   VAR
      sUDT_CommonStatus { ExternalAccessible := 'False'; ExternalVisible := 'False'; ExternalWritable := 'False'; S7_SetPoint := 'False'} : "UDT_CommonStatus";   // Common status structure
      sUDT_CommonStatusOld { ExternalAccessible := 'False'; ExternalVisible := 'False'; ExternalWritable := 'False'; S7_SetPoint := 'False'} : "UDT_CommonStatus";   // Auxiliary status structure
      sUDT_HMIStatus { ExternalAccessible := 'False'; ExternalVisible := 'False'; ExternalWritable := 'False'; S7_SetPoint := 'False'} : "UDT_CaljanStatus";   // HMI status structure
      sUDT_PNDevice { ExternalAccessible := 'False'; ExternalVisible := 'False'; ExternalWritable := 'False'; S7_SetPoint := 'False'} : "UDT_PNDevice";   // PN device info structure
      sa_PNPortsStatus { ExternalAccessible := 'False'; ExternalVisible := 'False'; ExternalWritable := 'False'} : Array[1..8] of Bool;   // TRUE when specific port has an error
      R_TRIG_EnergySave {InstructionName := 'R_TRIG'; LibVersion := '1.0'; ExternalAccessible := 'False'; ExternalVisible := 'False'; ExternalWritable := 'False'; S7_SetPoint := 'False'} : R_TRIG;   // Rising edge for energy save
      R_TRIG_ConveyorUp {InstructionName := 'R_TRIG'; LibVersion := '1.0'; ExternalAccessible := 'False'; ExternalVisible := 'False'; ExternalWritable := 'False'; S7_SetPoint := 'False'} : R_TRIG;   // Rising edge of automatic active
      R_TRIG_ConveyorDown {InstructionName := 'R_TRIG'; LibVersion := '1.0'; ExternalAccessible := 'False'; ExternalVisible := 'False'; ExternalWritable := 'False'; S7_SetPoint := 'False'} : R_TRIG;   // Rising edge of automatic not active
      R_TRIG_NotHealthy {InstructionName := 'R_TRIG'; LibVersion := '1.0'; ExternalAccessible := 'False'; ExternalVisible := 'False'; ExternalWritable := 'False'; S7_SetPoint := 'False'} : R_TRIG;   // Rising edge trigger if extendable not healthy
      R_TRIG_TooLongParcel {InstructionName := 'R_TRIG'; LibVersion := '1.0'; ExternalAccessible := 'False'; ExternalVisible := 'False'; ExternalWritable := 'False'; S7_SetPoint := 'False'} : R_TRIG;   // Rising edge trigger for too long parcel
      R_TRIG_SafetyOk {InstructionName := 'R_TRIG'; LibVersion := '1.0'; ExternalAccessible := 'False'; ExternalVisible := 'False'; ExternalWritable := 'False'; S7_SetPoint := 'False'} : R_TRIG;   // Rising edge trigger safety is ok
      R_TRIG_PEC_UnloaderFiltered {InstructionName := 'R_TRIG'; LibVersion := '1.0'; ExternalAccessible := 'False'; ExternalVisible := 'False'; ExternalWritable := 'False'; S7_SetPoint := 'False'} : R_TRIG;   // Rising edge trigger end of section photo eye filtered
      F_TRIG_PEC_UnloaderFiltered {InstructionName := 'F_TRIG'; LibVersion := '1.0'; ExternalAccessible := 'False'; ExternalVisible := 'False'; ExternalWritable := 'False'; S7_SetPoint := 'False'} : F_TRIG;   // Falling edge trigger end of section photo eye filtered
      F_TRIG_AuxHeadToEnd {InstructionName := 'F_TRIG'; LibVersion := '1.0'; ExternalAccessible := 'False'; ExternalVisible := 'False'; ExternalWritable := 'False'; S7_SetPoint := 'False'} : F_TRIG;   // Falling edge trigger Aux head to end bit
      R_TRIG_TailToBegin {InstructionName := 'R_TRIG'; LibVersion := '1.0'; ExternalAccessible := 'False'; ExternalVisible := 'False'; ExternalWritable := 'False'; S7_SetPoint := 'False'} : R_TRIG;   // Rising edge trigger tail to begin bit
      sR_TRIG_PNSlaveError {InstructionName := 'R_TRIG'; LibVersion := '1.0'; ExternalAccessible := 'False'; ExternalVisible := 'False'; ExternalWritable := 'False'; S7_SetPoint := 'False'} : R_TRIG;   // Rising edge for PN error
      sR_TRIG_PNSlaveNotOnline {InstructionName := 'R_TRIG'; LibVersion := '1.0'; ExternalAccessible := 'False'; ExternalVisible := 'False'; ExternalWritable := 'False'; S7_SetPoint := 'False'} : R_TRIG;   // Rising edge for PN not online
      sFB_PEC { ExternalAccessible := 'False'; ExternalVisible := 'False'; ExternalWritable := 'False'; S7_SetPoint := 'False'} : "FB_PEC";   // FB PEC block for PEC Jam status
      sFB_ResetPulseTimer { ExternalAccessible := 'False'; ExternalVisible := 'False'; ExternalWritable := 'False'; S7_SetPoint := 'False'} : "FB_TimerOnOffDelay";   // Timer on/off delay for reset pulse
      sFB_CascadeModeTimer { ExternalAccessible := 'False'; ExternalVisible := 'False'; ExternalWritable := 'False'; S7_SetPoint := 'False'} : "FB_TimerOnOffDelay";   // Timer on/off delay for cascade mode
      sFB_TimerOnOffDelayCheck24V { ExternalAccessible := 'False'; ExternalVisible := 'False'; ExternalWritable := 'False'; S7_SetPoint := 'False'} : "FB_TimerOnOffDelay";   // Timer on/off delay to allow startup before fault is generated
      sFB_TimerOnOffDelayCheck400V { ExternalAccessible := 'False'; ExternalVisible := 'False'; ExternalWritable := 'False'; S7_SetPoint := 'False'} : "FB_TimerOnOffDelay";   // Timer on/off delay to allow startup before fault is generated
      sFB_Displacement { ExternalAccessible := 'False'; ExternalVisible := 'False'; ExternalWritable := 'False'; S7_SetPoint := 'False'} : "FB_Displacement";   // Function block to calculate displacement
      sdi_GapHeadToHeadConfiguration { ExternalAccessible := 'False'; ExternalVisible := 'False'; ExternalWritable := 'False'} : DInt;   // Preset forward gap head to head with correction [cm]
      sdi_GapTailToHeadConfiguration { ExternalAccessible := 'False'; ExternalVisible := 'False'; ExternalWritable := 'False'} : DInt;   // Preset forward gap tail to head with correction [cm]
   END_VAR
   VAR RETAIN
      sdi_HeadToEnd { ExternalAccessible := 'False'; ExternalVisible := 'False'; ExternalWritable := 'False'} : DInt;   // Count head to end distance
      sdi_GapHeadToHead { ExternalAccessible := 'False'; ExternalVisible := 'False'; ExternalWritable := 'False'} : DInt;   // Head to head between two products
      sdi_TailToBegin { ExternalAccessible := 'False'; ExternalVisible := 'False'; ExternalWritable := 'False'} : DInt;   // Count tail to next conveyor distance
      sdi_AuxGapHeadToHeadCounter { ExternalAccessible := 'False'; ExternalVisible := 'False'; ExternalWritable := 'False'} : DInt;   // Auxiliary variable to count the head to head
      sdi_AuxGapTailtoHeadCounter { ExternalAccessible := 'False'; ExternalVisible := 'False'; ExternalWritable := 'False'} : DInt;   // Auxiliary variable to count the gap
      sdi_Gap { ExternalAccessible := 'False'; ExternalVisible := 'False'; ExternalWritable := 'False'} : DInt;   // Gap between two products
   END_VAR
   VAR
      si_AuxEnergySave { ExternalAccessible := 'False'; ExternalVisible := 'False'; ExternalWritable := 'False'} : Int;   // Auxiliary energy save
      sx_Disabled { ExternalAccessible := 'False'; ExternalVisible := 'False'; ExternalWritable := 'False'} : Bool;   // Operation is enabled
      sx_Ready { ExternalAccessible := 'False'; ExternalVisible := 'False'; ExternalWritable := 'False'} : Bool;   // Conveyor Ready to operate in Forward mode
      sx_PEC_EoSFiltered { ExternalAccessible := 'False'; ExternalVisible := 'False'; ExternalWritable := 'False'} : Bool;   // End of section photo eye filtered
      sx_EnergySaveActive { ExternalAccessible := 'False'; ExternalVisible := 'False'; ExternalWritable := 'False'} : Bool;   // Active energy save mode
      sx_AutomaticActive { ExternalAccessible := 'False'; ExternalVisible := 'False'; ExternalWritable := 'False'} : Bool;   // Forward active
      sx_CascadeStartUp { ExternalAccessible := 'False'; ExternalVisible := 'False'; ExternalWritable := 'False'} : Bool;   // Cascade startup auxiliary bit
      sx_ReverseActive { ExternalAccessible := 'False'; ExternalVisible := 'False'; ExternalWritable := 'False'} : Bool;   // Unloader is running in reverse directon
   END_VAR
   VAR RETAIN
      sx_AuxHeadToEnd { ExternalAccessible := 'False'; ExternalVisible := 'False'; ExternalWritable := 'False'} : Bool;   // Aux bit to control head to end positioning in forward direction
      sx_AuxHeadAtEnd { ExternalAccessible := 'False'; ExternalVisible := 'False'; ExternalWritable := 'False'} : Bool;   // Parcel reach the end of the conveyor in forward direction
      sx_Gapping { ExternalAccessible := 'False'; ExternalVisible := 'False'; ExternalWritable := 'False'} : Bool;   // Gapping in process in forward direction
      sx_TailToBegin { ExternalAccessible := 'False'; ExternalVisible := 'False'; ExternalWritable := 'False'} : Bool;   // Tail to begin done in forward direction
      sx_RecoveryGap { ExternalAccessible := 'False'; ExternalVisible := 'False'; ExternalWritable := 'False'} : Bool;   // Recovery gap activated in forward direction
   END_VAR
   VAR
      sx_HoldUnloading { ExternalAccessible := 'False'; ExternalVisible := 'False'; ExternalWritable := 'False'} : Bool;   // Hold unloading ofter release Hold Reverse button
      sx_24VOk { ExternalAccessible := 'False'; ExternalVisible := 'False'; ExternalWritable := 'False'} : Bool;   // 24V ok
      sx_400VOk { ExternalAccessible := 'False'; ExternalVisible := 'False'; ExternalWritable := 'False'} : Bool;   // 400V ok
   END_VAR

   VAR CONSTANT
      ci_OverflowLimit : Int := 32000;   // Limit int overflow
      ci_NumberOfProfinetPorts : Int := 2;   // Number of Profinet ports in device
      ci_PowerSupplyDelayTime : UInt := 4000;   // Power supply delay time
   END_VAR


BEGIN
	(*
	----------------------------------------------------------------------------------------

	Version history:
	Date        | Version   | Author        | Remark
	----------------------------------------------------------------------------------------
	26/10/2021  | 0.1       | M. Piela      | first release MHS TIA 16
	11/11/2021  | 0.2       | S. Theocharis | change profinet ok to hardware ok
	10/01/2022  | 0.3       | K. Pokorski   | Bug fix/PNPN coupler handling added
	21/02/2022  | 0.4       | M. Piela      | Status update
	12/03/2022  | 0.5       | M. Piela      | Add reset energy save via handshake
	09/05/2022  | 0.6       | M. Piela      | Correct contitions to allow loading and unloading
	24/06/2022  | 0.7       | M. Kurpiers   | Loader running and dieback status changed
	27/07/2022  | 0.8       | M. Piela      | Change conditon to energy save for loader
	21/02/2023  | 4.0       | F.Baten       | 4.0 Release TIA 17.5
	*)

	REGION 1 - Get Device Profinet information

	    "FC_GetDevicePN"(is_PNDeviceName := #iUDT_CaljanConfiguration.PNDeviceName,
	                     ix_SimulationModeActive := #ix_SimulationModeActive,
	                     iqUDT_PND := #sUDT_PNDevice);

	    "FC_GetPNPortStatus"(ii_NumberOfPorts := #ci_NumberOfProfinetPorts,
	                         iUDT_DevicePNInfo := #sUDT_PNDevice,
	                         qa_PortFault => #sa_PNPortsStatus);

	END_REGION

	REGION 2 - Initial

	    REGION 2.1 - First PLC cycle

	        IF "DB_Memory".FirstScan
	        THEN
	            #sx_AutomaticActive := FALSE;
	            #iqUDT_HandShakeUp.RTR := FALSE;
	            #iqUDT_HandShakeUp.CascadeStartUp := FALSE;
	            #sx_Disabled := FALSE;
	        END_IF;

	    END_REGION

	    REGION 2.2 - Triggers

	        // Rising edge trigger energy save
	        #R_TRIG_EnergySave(CLK := #sUDT_CommonStatus.EnergySave);

	        // Rising edge extendable up
	        #R_TRIG_ConveyorUp(CLK := #sx_AutomaticActive AND #sx_Ready);

	        // Rising edge extendable down
	        #R_TRIG_ConveyorDown(CLK := #sx_AutomaticActive AND NOT #sx_Ready);

	        // Rising edge extendable not healthy
	        #R_TRIG_NotHealthy(CLK := #sUDT_HMIStatus.Specific.NotHealthy);

	        // Rising edge for too long parcel
	        #R_TRIG_TooLongParcel(CLK := #sUDT_HMIStatus.Specific.TooLongParcel);

	        // Rising edge for Profinet error
	        #sR_TRIG_PNSlaveError(CLK := #sUDT_HMIStatus.Specific.PNSlaveError);

	        // Rising edge for Profinet not online
	        #sR_TRIG_PNSlaveNotOnline(CLK := #sUDT_HMIStatus.Specific.PNSlaveNotOnline);

	    END_REGION

	    REGION 2.3 - HMI button Disable operation

	        // Copy HMI command to static memory
	        #sx_Disabled := #iqUDT_CaljanCommand.Disable;

	        // Copy status to HMI
	        #sUDT_HMIStatus.Specific.Disabled := #sx_Disabled;

	    END_REGION

	    REGION 2.4 - Displacement

	        // Calculate displacement only when Caljan is running
	        IF #iUDT_CaljanReceive.BeltDirection_Loading OR #iUDT_CaljanReceive.BeltDirection_Unloading
	        THEN
	            #sFB_Displacement(#iqUDT_CaljanInterface);
	        ELSE
	            #iqUDT_CaljanInterface.Displacement := 0;
	        END_IF;

	        // Map displacement to upstream conveyor
	        IF NOT #sx_ReverseActive
	        THEN
	            #iqUDT_HandShakeUp.DownstreamDisplacement := #iqUDT_CaljanInterface.Displacement;
	        ELSE
	            #iqUDT_HandShake.DownstreamDisplacement := #iqUDT_CaljanInterface.Displacement;
	        END_IF;

	    END_REGION

	    REGION 2.5 - Gaps configuration

	        // Forward head to head
	        #sdi_GapHeadToHeadConfiguration := #iUDT_CaljanConfiguration.Forward_Direction.GapHeadToHead + #iUDT_CaljanConfiguration.Forward_Direction.GapCorrection;
	        // Forward tail to head
	        #sdi_GapTailToHeadConfiguration := #iUDT_CaljanConfiguration.Forward_Direction.GapTailToHead + #iUDT_CaljanConfiguration.Forward_Direction.GapCorrection;

	    END_REGION

	    REGION 2.6 - Timers

	        // Handle PEC when Calian is configured as unloader
	        IF #iUDT_CaljanConfiguration.CaljanMode = 2
	        THEN
	            // PEC EoS
	            #sFB_PEC(ix_PEC := #iUDT_CaljanReceive.PECUnloader,
	                     iUDT_PECConfiguration := #iUDT_CaljanConfiguration.PEC_EOS,
	                     qx_PECFiltered => #sx_PEC_EoSFiltered,
	                     qUDT_HMIStatus => #sUDT_HMIStatus.Specific.PEC_EoS,
	                     iqUDT_ConveyorInterface := #iqUDT_CaljanInterface,
	                     iqUDT_PECStatistics := #iqUDT_Statistics.PEC_EOS);
	        END_IF;

	        // Hardware will only be available after the delay, so the device has time for the initialisation
	        #sFB_TimerOnOffDelayCheck24V(iudi_OnDelayTime := #ci_PowerSupplyDelayTime,
	                                     ix_SignalToDelay := #ix_24vOk,
	                                     qx_DelayedSignal => #sx_24VOk);

	        #sFB_TimerOnOffDelayCheck400V(iudi_OnDelayTime := #ci_PowerSupplyDelayTime,
	                                      ix_SignalToDelay := #ix_400vOk,
	                                      qx_DelayedSignal => #sx_400VOk);

	    END_REGION

	END_REGION

	REGION 3 - Reset Profinet errors

	    IF #iqUDT_EquipmentControl.Command.Reset THEN
	        #sUDT_HMIStatus.Specific.PNSlaveNotOnline := FALSE;
	        #sUDT_HMIStatus.Specific.PNSlaveError := FALSE;
	        #sUDT_HMIStatus.Specific.PNSlaveWarning := FALSE;
	    END_IF;

	END_REGION

	REGION 4 - Errors

	    // Check if PN device is online
	    IF NOT "DB_ProfinetDiagnostic".ProfinetNetworks[#sUDT_PNDevice.PNNetworknumber].DeviceStatus[#sUDT_PNDevice.PNDeviceNumber].DeviceState.Exist
	        AND NOT #ix_SimulationModeActive
	        AND #sx_24VOk
	    THEN
	        #sUDT_HMIStatus.Specific.PNSlaveNotOnline := TRUE;

	    END_IF;

	    // Check if PN ports are healthy
	    IF #sa_PNPortsStatus[1] XOR #sa_PNPortsStatus[2] THEN
	        #sUDT_HMIStatus.Specific.PNSlaveWarning := TRUE;
	    END_IF;

	    // Check if PN device has an error
	    IF "DB_ProfinetDiagnostic".ProfinetNetworks[#sUDT_PNDevice.PNNetworknumber].DeviceStatus[#sUDT_PNDevice.PNDeviceNumber].DeviceState.Error
	        AND NOT #ix_SimulationModeActive
	        AND #sx_24VOk
	        AND NOT #sUDT_HMIStatus.Specific.PNSlaveWarning
	    THEN
	        #sUDT_HMIStatus.Specific.PNSlaveError := TRUE;
	    END_IF;

	    // Not healthy
	    #sUDT_HMIStatus.Specific.NotHealthy := NOT #iUDT_CaljanReceive.Healthy
	    AND #sx_400VOk
	    AND #sx_24VOk
	    AND #ix_HardwareOK
	    AND #ix_SafetyOk;

	    // Common Error
	    #sUDT_CommonStatus.Error := NOT #sx_24VOk
	    OR NOT #sx_400VOk
	    OR NOT #ix_HardwareOK
	    OR NOT #ix_SafetyOk
	    OR #sUDT_HMIStatus.Specific.PEC_EoS.Jam
	    OR #sUDT_HMIStatus.Specific.NotHealthy;

	    //Parcel too long
	    #sUDT_HMIStatus.Specific.TooLongParcel := #ix_TooLongParcel;

	    // Warning
	    #sUDT_CommonStatus.Warning := #sUDT_HMIStatus.Specific.TooLongParcel;

	END_REGION

	REGION 5 - Check conditions to set caljan ready

	    #sx_Ready := NOT #sUDT_CommonStatus.Error;

	END_REGION

	REGION 6 - Stop caljan

	    IF NOT #iqUDT_EquipmentControl.Command.AutomaticOn
	        OR #sUDT_CommonStatus.Error
	    THEN
	        #sx_AutomaticActive := FALSE;
	        #qUDT_CaljanSend.AllowLoading := FALSE;
	        #qUDT_CaljanSend.AllowUnloading := FALSE;
	        #iqUDT_HandShakeUp.RTR := FALSE;
	        #iqUDT_HandShakeUp.CascadeStartUp := FALSE;
	    END_IF;

	END_REGION

	REGION 7 - Start automatic mode

	    // If start (one shot) is received from system, this is memorised until started in cascade. Later the unloader is started
	    IF #iqUDT_EquipmentControl.Command.Start
	        AND #sx_Ready
	    THEN
	        #sx_AutomaticActive := TRUE;
	    END_IF;

	    //Timer to cascade mode
	    #sFB_CascadeModeTimer(iudi_OnDelayTime := #iUDT_CaljanConfiguration.CascadeTimeOnDelay,
	                          ix_SignalToDelay := #sx_AutomaticActive,
	                          ix_Enable := #sx_Ready,
	                          qx_DelayedSignal => #sx_CascadeStartUp);

	    #iqUDT_HandShakeUp.CascadeStartUp := #sx_CascadeStartUp;                                     //TO CHECK ON SITE

	END_REGION

	REGION 8 - Automatic mode active

	    REGION 8.1 - Operation

	        (* *******LOADER ******** *)
	        IF #iUDT_CaljanConfiguration.CaljanMode = 1 THEN

	            // Release loading
	            #qUDT_CaljanSend.AllowLoading := #sx_AutomaticActive
	            AND #sx_Ready
	            AND #iUDT_CaljanReceive.ReadyToReceive
	            AND NOT #sx_Disabled
	            AND NOT #ix_ExternalRequestHold
	            AND NOT #sx_EnergySaveActive;

	            #iqUDT_HandShakeUp.RTR := #qUDT_CaljanSend.AllowLoading;

	        END_IF;

	        (* *******UNLOADER ******** *)
	        IF #iUDT_CaljanConfiguration.CaljanMode = 2
	        THEN

	            // Release unloading
	            #qUDT_CaljanSend.AllowUnloading := #sx_AutomaticActive
	            AND #sx_Ready
	            AND NOT #sx_Disabled
	            AND NOT #ix_ExternalRequestHold
	            AND NOT #sx_EnergySaveActive
	            AND NOT #sx_HoldUnloading;

	            #qUDT_CaljanSend.PEC_Override := #iqUDT_HandShake.RTR
	            AND NOT #ix_ExternalRequestDieBack;

	        END_IF;

	    END_REGION

	    REGION 8.2 - Energy save

	        IF #iUDT_CaljanConfiguration.Energy THEN

	            // Set Energy save active
	            IF #si_AuxEnergySave >= #iUDT_CaljanConfiguration.EnergySaveLength
	            THEN
	                #sx_EnergySaveActive := TRUE;
	            END_IF;

	            (* *******LOADER ******** *)
	            // Reset or increment displacement calculation to use for energy save
	            IF #iUDT_CaljanConfiguration.CaljanMode = 1
	                AND NOT #iUDT_CaljanReceive.PECUnloader
	                OR #ix_ResetEnergySave
	                OR #iqUDT_HandShakeUp.RTS
	                OR #iqUDT_HandShakeUp.ResetEnergySave
	                OR NOT #iqUDT_EquipmentControl.Command.AutomaticOn
	            THEN
	                #si_AuxEnergySave := 0;
	                #sx_EnergySaveActive := FALSE;

	                (* *******UNLOADER ******** *)
	            ELSIF #iUDT_CaljanConfiguration.CaljanMode = 2
	                AND NOT #sx_PEC_EoSFiltered
	                OR #ix_ResetEnergySave
	                OR #iUDT_CaljanReceive.HoldReverseSignal
	            THEN
	                #si_AuxEnergySave := 0;
	                #sx_EnergySaveActive := FALSE;

	            ELSE
	                #si_AuxEnergySave += #iqUDT_CaljanInterface.Displacement;
	            END_IF;
	        ELSE
	            #si_AuxEnergySave := 0;
	            #sx_EnergySaveActive := FALSE;

	        END_IF;

	        IF #sx_AutomaticActive AND NOT #sx_ReverseActive
	        THEN
	            #iqUDT_HandShake.ResetEnergySave := NOT #iUDT_CaljanReceive.PECUnloader AND NOT #sx_EnergySaveActive;
	        END_IF;

	    END_REGION

	END_REGION

	REGION 9 - Gapping configuration

	    REGION 9.1 - Head to End

	        (*  Function to calculate when the head of the parcel reaches the end of the conveyor
	            When PEC detects parcels head, the functionality increments the displacement of the conveyor until reach the value of the distance
	            between PEC and the end of the conveyor. After that, the counter is reset and the bit #sx_AuxHeadToEnd is triggered to inform the system. *)
	        IF NOT #sx_ReverseActive
	        THEN
	            REGION 9.1.1 - Forward

	                #F_TRIG_PEC_UnloaderFiltered(CLK := #sx_PEC_EoSFiltered);

	                IF #F_TRIG_PEC_UnloaderFiltered.Q                                   // Detects the product's head
	                THEN
	                    #sdi_HeadToEnd := #iUDT_CaljanConfiguration.PEC_EOS.Distance;  // move the distance between PEC and the end of the conveyor to auxiliary variable
	                    #sx_AuxHeadToEnd := TRUE;                                       // Active head to end function

	                    #sdi_GapHeadToHead := #sdi_AuxGapHeadToHeadCounter;             // Move gap calculated to variable
	                    #sdi_AuxGapHeadToHeadCounter := 0;                              // Reset gap counter

	                    #sdi_Gap := #sdi_AuxGapTailtoHeadCounter;                       // Move gap calculated to variable

	                    #sdi_AuxGapTailtoHeadCounter := 0;                              // Reset gap counter

	                    #iqUDT_HandShake.RTS := TRUE;                                  // Set ready to send true when a parcel is detected in the PEC
	                END_IF;

	                IF #sx_AuxHeadToEnd                                                 // Parcel's head detected in photo cell
	                    AND (#sdi_HeadToEnd > 0)                                        // Psrcel's head do not arrive in the end of the conveyor yet
	                THEN
	                    #sdi_HeadToEnd -= #iqUDT_CaljanInterface.Displacement;         // Count displacement until arrive to the end of the conveyor
	                ELSE
	                    #sx_AuxHeadToEnd := FALSE;                                      // Stop function head to end
	                END_IF;

	                // Falling edge trigger Aux Head to End bit
	                #F_TRIG_AuxHeadToEnd(CLK := #sx_AuxHeadToEnd);

	                IF #F_TRIG_AuxHeadToEnd.Q

	                THEN
	                    #sx_AuxHeadAtEnd := TRUE;                                       // The head of the parcel is at the front positon of the conveyor
	                END_IF;

	            END_REGION

	        END_IF;

	    END_REGION

	    REGION 9.2 - Tail to Begin

	        (*   This function tracks when parcels tail reaches the begin of downstream conveyor
	             When the PEC is clear, the function start to increase the displacement until reaches the distance
	             between PEC and the end of conveyor. *)
	        IF NOT #sx_ReverseActive
	        THEN
	            REGION 9.2.1 - Forward

	                #R_TRIG_PEC_UnloaderFiltered(CLK := #sx_PEC_EoSFiltered);

	                IF #R_TRIG_PEC_UnloaderFiltered.Q                                             // Detects product's tail
	                THEN

	                    #sdi_TailToBegin := (#iUDT_CaljanConfiguration.PEC_EOS.Distance / 10);   // move distance between PE and the end of the conveyor to auxiliar variable

	                END_IF;

	                IF (#sdi_TailToBegin > 0)                                                     // While tails parcel do not reach the beginning of next conveyor
	                THEN

	                    #sdi_TailToBegin -= #iqUDT_CaljanInterface.Displacement;                 // count displacement until the product's tail arrive to the next conveyor
	                    #sx_TailToBegin := FALSE;                                                 // Reset tail to begin bit

	                ELSE

	                    #sx_TailToBegin := TRUE;                                                  // Product's tail arrived at the begin OF next conveyor

	                END_IF;

	                // Rising edge trigger Aux tail to Begin bit
	                #R_TRIG_TailToBegin(CLK := #sx_TailToBegin);

	            END_REGION

	        END_IF;

	    END_REGION

	    REGION 9.3 - Gap

	        (*    Gap tail TO head function calculates the distance (Gap) between two parcels.
	              The function increases the Counter WHILE the photo eye is clear.
	              Every time a parcel trigger the photo eye, gap value is save AND the counter is reset.  *)
	        IF NOT #sx_ReverseActive
	        THEN
	            REGION 9.3.1 - Forward

	                IF #iUDT_CaljanReceive.PECUnloader                             // Count displacement when the PE do not detects the product
	                THEN

	                    IF #sdi_AuxGapTailtoHeadCounter < #ci_OverflowLimit        // Prevent integer variable overflow
	                    THEN
	                        IF #iqUDT_HandShake.RTR THEN
	                            #sdi_AuxGapTailtoHeadCounter += #iqUDT_CaljanInterface.Displacement;    // Calculate the gap
	                        END_IF;

	                    END_IF;

	                END_IF;

	            END_REGION

	        END_IF;

	    END_REGION

	    REGION 9.4 - Head to head

	        // The functionality head to head is used to calculate the distance between one head's parcel and the head's parcel behind.
	        // To do it, everytime the PEC is triggered, the function save the distance calculated and reset the counter to start
	        // counting again, over and over again.
	        IF NOT #sx_ReverseActive
	        THEN
	            REGION 9.4.1 - Forward

	                IF #sdi_AuxGapHeadToHeadCounter < #ci_OverflowLimit                         // Prevent integer variable overflow
	                THEN

	                    #sdi_AuxGapHeadToHeadCounter += #iqUDT_CaljanInterface.Displacement;   // measure the distance between two products

	                END_IF;

	            END_REGION

	        END_IF;

	    END_REGION

	    REGION 9.5 - Check gaps between products

	        // Check gaps is a routine that checks all the time if the gap and head to head distance is acording to the configuration.
	        // If not, the bit "sx_Gapping" is set true and the conveyor stops to gap.
	        // Compare gaps calculated with the configured gaps
	        IF NOT #sx_ReverseActive
	        THEN
	            REGION 9.5.1 - Forward

	                IF ((#sdi_GapHeadToHeadConfiguration > #sdi_GapHeadToHead        // Compare head to head configured with real distance
	                    OR #sdi_GapTailToHeadConfiguration > #sdi_Gap)
	                    AND #F_TRIG_AuxHeadToEnd.Q)                                  // Trigger when parcel arrive in the end of the conveyor
	                THEN

	                    #sx_Gapping := TRUE;        // Bit to inform the system that conveyor needs to stop to apply gap

	                END_IF;

	            END_REGION

	        END_IF;
	        //    When conveyor stops to gapping, displacement values from downstream are used to
	        //    apply new gap.
	        //    When the new gap applied fits with the configured one, the conveyor starts running again.
	        //    If the conveyor stops for die back reason and the gap its been applied, and extra gap value it will be applied.
	        //    This recovery gap it helps to recovery the system after die back.
	        IF NOT #sx_ReverseActive
	        THEN
	            REGION 9.5.2 - Forward recovery

	                IF (#sx_Gapping                                                   // Gapping needs to be applied bit
	                    AND ((#sdi_GapHeadToHeadConfiguration > #sdi_GapHeadToHead    // Configured head to head bigger than the actual one
	                    OR #sdi_GapTailToHeadConfiguration > #sdi_Gap)                // Configured gap bigger than the actual one
	                    AND NOT #sx_RecoveryGap)                                      // Die back recovery gap bit not active
	                    OR ((#sdi_GapHeadToHeadConfiguration > #sdi_GapHeadToHead     // Actual head to head distance
	                    OR #sdi_GapTailToHeadConfiguration > #sdi_Gap)                // Actual gap between parcels
	                    AND #sx_RecoveryGap))                                         // Recovery gap bit activate
	                THEN

	                    #sdi_GapHeadToHead += #iqUDT_HandShake.DownstreamDisplacement;     // Increase head to head counter with conveyor downstream displacement
	                    #sdi_Gap += #iqUDT_HandShake.DownstreamDisplacement;               // Increase gap counter with conveyor downstream displacement

	                ELSE

	                    #sx_Gapping := FALSE;          // Set gapping bit to false

	                END_IF;

	                IF #sx_Gapping                     // Gapping bit active
	                    AND NOT #iqUDT_HandShake.RTR  // Ready to receive not active
	                THEN

	                    #sx_RecoveryGap := TRUE;       // Recovery gap activation after die back

	                END_IF;

	                IF #sx_RecoveryGap                 // Recovery gap active
	                    AND NOT #sx_Gapping            // Gapping bit not active
	                THEN

	                    #sx_RecoveryGap := FALSE;      // Recovery gap disable

	                END_IF;

	            END_REGION

	        END_IF;

	    END_REGION

	    REGION 9.6 - Ready to send and Transfer in progress

	        IF NOT #sx_ReverseActive
	        THEN
	            REGION 9.6.1 - Forward

	                IF #iqUDT_HandShake.RTR                 // Ready to receive bit
	                    AND #iqUDT_HandShakeUp.RTR
	                    AND NOT #sx_Gapping
	                    AND #sx_AuxHeadAtEnd                 // Parcel is at end of conveyor
	                    AND NOT #ix_ExternalRequestDieBack
	                THEN

	                    #iqUDT_HandShake.TIP := TRUE;      // Transfer in progress bit
	                    #iqUDT_HandShake.RTS := FALSE;     // Ready to send bit
	                    #sx_AuxHeadAtEnd := FALSE;

	                END_IF;

	                IF #R_TRIG_TailToBegin.Q               // Reset TIP when the parcel leaves interlock
	                THEN

	                    #iqUDT_HandShake.TIP := FALSE;     // Transfer in progress bit

	                END_IF;

	            END_REGION

	        END_IF;

	    END_REGION

	END_REGION

	REGION 10 - Reverse run

	    IF #iUDT_CaljanConfiguration.CaljanMode = 2 THEN

	        //Starting reverse run
	        IF #iUDT_CaljanReceive.HoldReverseSignal
	            AND #sx_AutomaticActive
	        THEN
	            #sx_ReverseActive := TRUE;
	        END_IF;

	        IF #sx_ReverseActive AND NOT #iUDT_CaljanReceive.HoldReverseSignal
	        THEN
	            #sx_ReverseActive := FALSE;
	            #sx_HoldUnloading := TRUE;
	        END_IF;

	        IF NOT #iUDT_CaljanReceive.HoldReverseSignal AND #iUDT_CaljanReceive.ResetReverse
	        THEN
	            #sx_ReverseActive := FALSE;
	            #sx_HoldUnloading := FALSE;
	        END_IF;
	    END_IF;

	END_REGION

	REGION 11 - Reset

	    // Safety ok extended pulse
	    #R_TRIG_SafetyOk(CLK := #ix_SafetyReset);

	    #sFB_ResetPulseTimer(iudi_OffDelayTime := #iUDT_CaljanConfiguration.ResetDelay,
	                         ix_SignalToDelay := #R_TRIG_SafetyOk.Q);

	    // Send reset signal to Caljan
	    #qUDT_CaljanSend.Reset := #ix_SafetyReset OR #iqUDT_EquipmentControl.Command.Reset OR #sFB_ResetPulseTimer.qx_DelayedSignal;

	END_REGION

	REGION 12 - Status

	    #sUDT_CommonStatus.Stopped := NOT #sx_AutomaticActive;
	    #sUDT_CommonStatus.Running := (#iUDT_CaljanReceive.BeltDirection_Unloading OR #iUDT_CaljanReceive.BeltDirection_Loading) AND #iUDT_CaljanReceive.ActualSpeed > 0;
	    #sUDT_CommonStatus.AutoON := #sx_Ready AND #sx_AutomaticActive;
	    #sUDT_CommonStatus.Halted := #ix_ExternalRequestHold AND #sUDT_CommonStatus.AutoON AND NOT #sx_EnergySaveActive;
	    #sUDT_CommonStatus.Dieback := (NOT #iqUDT_HandShake.RTR OR #ix_ExternalRequestDieBack) AND #sUDT_CommonStatus.AutoON AND NOT #sx_EnergySaveActive
	    AND NOT #sUDT_CommonStatus.EnergySave AND NOT #sUDT_CommonStatus.Running AND NOT #sx_PEC_EoSFiltered;

	    #sUDT_CommonStatus.EnergySave := #sx_EnergySaveActive;
	    #sUDT_CommonStatus.SafetyStop := NOT #ix_SafetyOk;

	    // HMI status update on change
	    IF #sUDT_CommonStatusOld <> #sUDT_CommonStatus
	    THEN
	        // HMI status initialization
	        #sUDT_HMIStatus.Status := 0;

	        // Running
	        IF #sUDT_CommonStatus.Running
	        THEN
	            #sUDT_HMIStatus.Status := "DB_HMIStatusConfiguration".Running;
	        END_IF;

	        // Stopped
	        IF #sUDT_CommonStatus.Stopped
	        THEN
	            #sUDT_HMIStatus.Status := "DB_HMIStatusConfiguration".Stopped;
	        END_IF;

	        // Energy save
	        IF #sUDT_CommonStatus.EnergySave
	        THEN
	            #sUDT_HMIStatus.Status := "DB_HMIStatusConfiguration".EnergySave;
	        END_IF;

	        // Dieback
	        IF #sUDT_CommonStatus.Dieback
	        THEN
	            #sUDT_HMIStatus.Status := "DB_HMIStatusConfiguration".Dieback;
	        END_IF;

	        // Halted
	        IF #sUDT_CommonStatus.Halted
	        THEN
	            #sUDT_HMIStatus.Status := "DB_HMIStatusConfiguration".Halted;
	        END_IF;

	        // Dimension error
	        IF #sUDT_HMIStatus.Specific.TooLongParcel
	        THEN
	            #sUDT_HMIStatus.Status := "DB_HMIStatusConfiguration".DimensionError;
	        END_IF;

	        //  PEC error
	        IF #sUDT_HMIStatus.Specific.PEC_EoS.Jam
	        THEN
	            #sUDT_HMIStatus.Status := "DB_HMIStatusConfiguration".PECJam;
	        END_IF;

	        // Not healthy
	        IF #sUDT_HMIStatus.Specific.NotHealthy
	        THEN
	            #sUDT_HMIStatus.Status := "DB_HMIStatusConfiguration".VFDNotHealthy;
	        END_IF;

	        // Safety stop
	        IF #sUDT_CommonStatus.SafetyStop
	        THEN
	            #sUDT_HMIStatus.Status := "DB_HMIStatusConfiguration".SafetyStop;
	        END_IF;

	        // Copy statuses

	        #sUDT_CommonStatusOld := #sUDT_CommonStatus;
	        #qUDT_Status := #sUDT_CommonStatus;
	    END_IF;

	    #qUDT_HMIStatus := #sUDT_HMIStatus;

	END_REGION

	REGION 13 - Statistics

	    // Up time
	    IF #sx_AutomaticActive
	        AND #sx_Ready
	        OR #iqUDT_EquipmentControl.Command.ResetData
	    THEN
	        "FC_Statistics"(ix_Reset := #iqUDT_EquipmentControl.Command.ResetData,
	                        ix_Activate := #sx_AutomaticActive AND #sx_Ready,
	                        ix_RTrigActivate := #R_TRIG_ConveyorUp.Q,
	                        iqUDT_Statistics := #iqUDT_Statistics.ExtendableUpTime);
	    END_IF;

	    // Down time
	    IF NOT #sx_AutomaticActive
	        AND #sx_Ready
	        OR #iqUDT_EquipmentControl.Command.ResetData
	    THEN
	        "FC_Statistics"(ix_Reset := #iqUDT_EquipmentControl.Command.ResetData,
	                        ix_Activate := NOT #sx_AutomaticActive AND #sx_Ready,
	                        ix_RTrigActivate := #R_TRIG_ConveyorDown.Q,
	                        iqUDT_Statistics := #iqUDT_Statistics.ExtendableDownTime);
	    END_IF;

	    // Energy save mode active
	    IF #sx_EnergySaveActive
	        OR #iqUDT_EquipmentControl.Command.ResetData
	    THEN
	        "FC_Statistics"(ix_Reset := #iqUDT_EquipmentControl.Command.ResetData,
	                        ix_Activate := #sUDT_CommonStatus.EnergySave,

	                        ix_RTrigActivate := #R_TRIG_EnergySave.Q,
	                        iqUDT_Statistics := #iqUDT_Statistics.EnergySave);
	    END_IF;

	    // Not healthy
	    IF #sUDT_HMIStatus.Specific.NotHealthy
	        OR #iqUDT_EquipmentControl.Command.ResetData
	    THEN
	        "FC_Statistics"(ix_Reset := #iqUDT_EquipmentControl.Command.ResetData,
	                        ix_Activate := #sUDT_HMIStatus.Specific.NotHealthy,
	                        ix_RTrigActivate := #R_TRIG_NotHealthy.Q,
	                        iqUDT_Statistics := #iqUDT_Statistics.NotHealthy);
	    END_IF;

	    // Too long parcel
	    IF #sUDT_HMIStatus.Specific.TooLongParcel
	        OR #iqUDT_EquipmentControl.Command.ResetData
	    THEN
	        "FC_Statistics"(ix_Reset := #iqUDT_EquipmentControl.Command.ResetData,
	                        ix_Activate := #sUDT_HMIStatus.Specific.TooLongParcel,
	                        ix_RTrigActivate := #R_TRIG_TooLongParcel.Q,
	                        iqUDT_Statistics := #iqUDT_Statistics.TooLongParcel);
	    END_IF;

	    // PN Slave not online
	    IF #iqUDT_EquipmentControl.Command.ResetData OR #sUDT_HMIStatus.Specific.PNSlaveNotOnline
	    THEN

	        "FC_Statistics"(ix_Reset := #iqUDT_EquipmentControl.Command.ResetData,
	                        ix_Activate := #sUDT_HMIStatus.Specific.PNSlaveNotOnline,
	                        ix_RTrigActivate := #sR_TRIG_PNSlaveNotOnline.Q,
	                        iqUDT_Statistics := #iqUDT_Statistics.PNNodeNotOnline);
	    END_IF;

	    // PN Slave error
	    IF #iqUDT_EquipmentControl.Command.ResetData OR #sUDT_HMIStatus.Specific.PNSlaveError
	    THEN

	        "FC_Statistics"(ix_Reset := #iqUDT_EquipmentControl.Command.ResetData,
	                        ix_Activate := #sUDT_HMIStatus.Specific.PNSlaveError,
	                        ix_RTrigActivate := #sR_TRIG_PNSlaveError.Q,
	                        iqUDT_Statistics := #iqUDT_Statistics.PNNodeError);
	    END_IF;

	END_REGION

	REGION 14 - Report to control block

	    "FC_EquipmentReport"(iUDT_Status := #sUDT_CommonStatus,
	                         iqUDT_Control := #iqUDT_EquipmentControl);

	END_REGION
END_FUNCTION_BLOCK

FUNCTION_BLOCK "FB_PowerDistributionPanel"
TITLE = PDP Block
{ S7_Optimized_Access := 'TRUE' }
AUTHOR : MHSE
VERSION : 3.0
// ATTRIBUTES
// AUTO_NUMBER = True
// BLOCK_NUMBER = 24
// END_ATTRIBUTES
   VAR_INPUT
      ix_24VOk { ExternalAccessible := 'False'; ExternalVisible := 'False'; ExternalWritable := 'False'} : Bool;   //  24VDC input OK
      ix_ET200Ok { ExternalAccessible := 'False'; ExternalVisible := 'False'; ExternalWritable := 'False'} : Bool;   //  ET 200 OK
      ix_CircuitBreakerOkF100 { ExternalAccessible := 'False'; ExternalVisible := 'False'; ExternalWritable := 'False'} : Bool;   //  Circuit breaker ok when the signal is true
      ix_CircuitBreakerOkF201 { ExternalAccessible := 'False'; ExternalVisible := 'False'; ExternalWritable := 'False'} : Bool;   //  Circuit breaker ok when the signal is true
      ix_CircuitBreakerOkF202 { ExternalAccessible := 'False'; ExternalVisible := 'False'; ExternalWritable := 'False'} : Bool;   //  Circuit breaker ok when the signal is true
      ix_CircuitBreakerOkF203 { ExternalAccessible := 'False'; ExternalVisible := 'False'; ExternalWritable := 'False'} : Bool;   //  Circuit breaker ok when the signal is true
      ix_CircuitBreakerOkF204 { ExternalAccessible := 'False'; ExternalVisible := 'False'; ExternalWritable := 'False'} : Bool;   //  Circuit breaker ok when the signal is true
      ix_CircuitBreakerOkF205 { ExternalAccessible := 'False'; ExternalVisible := 'False'; ExternalWritable := 'False'} : Bool;   //  Circuit breaker ok when the signal is true
      ix_CircuitBreakerOkF206 { ExternalAccessible := 'False'; ExternalVisible := 'False'; ExternalWritable := 'False'} : Bool;   //  Circuit breaker ok when the signal is true
      ix_CircuitBreakerOkF207 { ExternalAccessible := 'False'; ExternalVisible := 'False'; ExternalWritable := 'False'} : Bool;   //  Circuit breaker ok when the signal is true
      ix_CircuitBreakerOkF208 { ExternalAccessible := 'False'; ExternalVisible := 'False'; ExternalWritable := 'False'} : Bool;   //  Circuit breaker ok when the signal is true
      ix_CircuitBreakerOkF209 { ExternalAccessible := 'False'; ExternalVisible := 'False'; ExternalWritable := 'False'} : Bool;   //  Circuit breaker ok when the signal is true
      ix_CircuitBreakerOkF210 { ExternalAccessible := 'False'; ExternalVisible := 'False'; ExternalWritable := 'False'} : Bool;   //  Circuit breaker ok when the signal is true
      ix_CircuitBreakerOkF211 { ExternalAccessible := 'False'; ExternalVisible := 'False'; ExternalWritable := 'False'} : Bool;   //  Circuit breaker ok when the signal is true
      ix_CircuitBreakerOkF212 { ExternalAccessible := 'False'; ExternalVisible := 'False'; ExternalWritable := 'False'} : Bool;   //  Circuit breaker ok when the signal is true
      ix_CircuitBreakerOkF213 { ExternalAccessible := 'False'; ExternalVisible := 'False'; ExternalWritable := 'False'} : Bool;   //  Circuit breaker ok when the signal is true
      ix_CircuitBreakerOkF214 { ExternalAccessible := 'False'; ExternalVisible := 'False'; ExternalWritable := 'False'} : Bool;   //  Circuit breaker ok when the signal is true
      ix_CircuitBreakerOkF215 { ExternalAccessible := 'False'; ExternalVisible := 'False'; ExternalWritable := 'False'} : Bool;   //  Circuit breaker ok when the signal is true
      ix_CircuitBreakerOkF216 { ExternalAccessible := 'False'; ExternalVisible := 'False'; ExternalWritable := 'False'} : Bool;   //  Circuit breaker ok when the signal is true
      ix_CircuitBreakerOkF217 { ExternalAccessible := 'False'; ExternalVisible := 'False'; ExternalWritable := 'False'} : Bool;   //  Circuit breaker ok when the signal is true
      ix_CircuitBreakerOkF218 { ExternalAccessible := 'False'; ExternalVisible := 'False'; ExternalWritable := 'False'} : Bool;   //  Circuit breaker ok when the signal is true
      ix_CircuitBreakerOkF219 { ExternalAccessible := 'False'; ExternalVisible := 'False'; ExternalWritable := 'False'} : Bool;   //  Circuit breaker ok when the signal is true
      ix_CircuitBreakerOkF220 { ExternalAccessible := 'False'; ExternalVisible := 'False'; ExternalWritable := 'False'} : Bool;   //  Circuit breaker ok when the signal is true
      ix_CircuitBreakerOkF221 { ExternalAccessible := 'False'; ExternalVisible := 'False'; ExternalWritable := 'False'} : Bool;   //  Circuit breaker ok when the signal is true
      ix_CircuitBreakerOkF222 { ExternalAccessible := 'False'; ExternalVisible := 'False'; ExternalWritable := 'False'} : Bool;   //  Circuit breaker ok when the signal is true
      ix_CircuitBreakerOkF223 { ExternalAccessible := 'False'; ExternalVisible := 'False'; ExternalWritable := 'False'} : Bool;   //  Circuit breaker ok when the signal is true
      ix_CircuitBreakerOkF224 { ExternalAccessible := 'False'; ExternalVisible := 'False'; ExternalWritable := 'False'} : Bool;   //  Circuit breaker ok when the signal is true
      ix_CircuitBreakerOkF225 { ExternalAccessible := 'False'; ExternalVisible := 'False'; ExternalWritable := 'False'} : Bool;   //  Circuit breaker ok when the signal is true
      ix_CircuitBreakerOkF226 { ExternalAccessible := 'False'; ExternalVisible := 'False'; ExternalWritable := 'False'} : Bool;   //  Circuit breaker ok when the signal is true
      ix_CircuitBreakerOkF227 { ExternalAccessible := 'False'; ExternalVisible := 'False'; ExternalWritable := 'False'} : Bool;   //  Circuit breaker ok when the signal is true
      ix_CircuitBreakerOkF228 { ExternalAccessible := 'False'; ExternalVisible := 'False'; ExternalWritable := 'False'} : Bool;   //  Circuit breaker ok when the signal is true
      ix_CircuitBreakerOkF229 { ExternalAccessible := 'False'; ExternalVisible := 'False'; ExternalWritable := 'False'} : Bool;   //  Circuit breaker ok when the signal is true
      ix_CircuitBreakerOkF230 { ExternalAccessible := 'False'; ExternalVisible := 'False'; ExternalWritable := 'False'} : Bool;   //  Circuit breaker ok when the signal is true
      ix_CircuitBreakerOkF231 { ExternalAccessible := 'False'; ExternalVisible := 'False'; ExternalWritable := 'False'} : Bool;   //  Circuit breaker ok when the signal is true
      ix_CircuitBreakerOkF232 { ExternalAccessible := 'False'; ExternalVisible := 'False'; ExternalWritable := 'False'} : Bool;   //  Circuit breaker ok when the signal is true
      ix_CircuitBreakerOkF233 { ExternalAccessible := 'False'; ExternalVisible := 'False'; ExternalWritable := 'False'} : Bool;   //  Circuit breaker ok when the signal is true
      ix_CircuitBreakerOkF234 { ExternalAccessible := 'False'; ExternalVisible := 'False'; ExternalWritable := 'False'} : Bool;   //  Circuit breaker ok when the signal is true
      ix_CircuitBreakerOkF235 { ExternalAccessible := 'False'; ExternalVisible := 'False'; ExternalWritable := 'False'} : Bool;   //  Circuit breaker ok when the signal is true
      ix_CircuitBreakerOkF236 { ExternalAccessible := 'False'; ExternalVisible := 'False'; ExternalWritable := 'False'} : Bool;   //  Circuit breaker ok when the signal is true
      ix_CircuitBreakerOkF237 { ExternalAccessible := 'False'; ExternalVisible := 'False'; ExternalWritable := 'False'} : Bool;   //  Circuit breaker ok when the signal is true
      ix_CircuitBreakerOkF238 { ExternalAccessible := 'False'; ExternalVisible := 'False'; ExternalWritable := 'False'} : Bool;   //  Circuit breaker ok when the signal is true
      ix_CircuitBreakerOkF239 { ExternalAccessible := 'False'; ExternalVisible := 'False'; ExternalWritable := 'False'} : Bool;   //  Circuit breaker ok when the signal is true
      ix_CircuitBreakerOkF240 { ExternalAccessible := 'False'; ExternalVisible := 'False'; ExternalWritable := 'False'} : Bool;   //  Circuit breaker ok when the signal is true
      ix_CircuitBreakerOkF241 { ExternalAccessible := 'False'; ExternalVisible := 'False'; ExternalWritable := 'False'} : Bool;   //  Circuit breaker ok when the signal is true
      ix_CircuitBreakerOkF242 { ExternalAccessible := 'False'; ExternalVisible := 'False'; ExternalWritable := 'False'} : Bool;   //  Circuit breaker ok when the signal is true
      ix_CircuitBreakerOkF243 { ExternalAccessible := 'False'; ExternalVisible := 'False'; ExternalWritable := 'False'} : Bool;   //  Circuit breaker ok when the signal is true
      ix_CircuitBreakerOkF244 { ExternalAccessible := 'False'; ExternalVisible := 'False'; ExternalWritable := 'False'} : Bool;   //  Circuit breaker ok when the signal is true
      ix_CircuitBreakerOkF245 { ExternalAccessible := 'False'; ExternalVisible := 'False'; ExternalWritable := 'False'} : Bool;   //  Circuit breaker ok when the signal is true
      ix_CircuitBreakerOkF246 { ExternalAccessible := 'False'; ExternalVisible := 'False'; ExternalWritable := 'False'} : Bool;   //  Circuit breaker ok when the signal is true
      ix_CircuitBreakerOkF247 { ExternalAccessible := 'False'; ExternalVisible := 'False'; ExternalWritable := 'False'} : Bool;   //  Circuit breaker ok when the signal is true
      ix_CircuitBreakerOkF248 { ExternalAccessible := 'False'; ExternalVisible := 'False'; ExternalWritable := 'False'} : Bool;   //  Circuit breaker ok when the signal is true
      ix_CircuitBreakerOkF249 { ExternalAccessible := 'False'; ExternalVisible := 'False'; ExternalWritable := 'False'} : Bool;   //  Circuit breaker ok when the signal is true
      ix_CircuitBreakerOkF250 { ExternalAccessible := 'False'; ExternalVisible := 'False'; ExternalWritable := 'False'} : Bool;   //  Circuit breaker ok when the signal is true
      ix_CircuitBreakerOkF501 { ExternalAccessible := 'False'; ExternalVisible := 'False'; ExternalWritable := 'False'} : Bool;   //  Circuit breaker ok when the signal is true
      ix_CircuitBreakerOkF502 { ExternalAccessible := 'False'; ExternalVisible := 'False'; ExternalWritable := 'False'} : Bool;   //  Circuit breaker ok when the signal is true
      ix_CircuitBreakerOkF503 { ExternalAccessible := 'False'; ExternalVisible := 'False'; ExternalWritable := 'False'} : Bool;   //  Circuit breaker ok when the signal is true
      ix_CircuitBreakerOkF504 { ExternalAccessible := 'False'; ExternalVisible := 'False'; ExternalWritable := 'False'} : Bool;   //  Circuit breaker ok when the signal is true
      ix_CircuitBreakerOkF505 { ExternalAccessible := 'False'; ExternalVisible := 'False'; ExternalWritable := 'False'} : Bool;   //  Circuit breaker ok when the signal is true
      ix_HardwareOk { ExternalAccessible := 'False'; ExternalVisible := 'False'; ExternalWritable := 'False'} : Bool;   //  TRUE when  hardware is Ok
   END_VAR

   VAR_OUTPUT
      qUDT_PdpCbState { ExternalAccessible := 'False'; ExternalVisible := 'False'; ExternalWritable := 'False'} : "UDT_PowerDistributionPanelCBState";   //  Circuit breakers state
      qUDT_HMIStatus { ExternalAccessible := 'False'; ExternalVisible := 'False'; ExternalWritable := 'False'} : "UDT_PowerDistributionPanelStatus";   //  HMI status structure
      qUDT_Status { ExternalAccessible := 'False'; ExternalVisible := 'False'; ExternalWritable := 'False'} : "UDT_CommonStatus";   //  Common status structure
   END_VAR

   VAR_IN_OUT
      iqUDT_EquipmentControl : "UDT_EquipmentControl";   //  User-defined structure of equipment control commands.
      iq_CircuitBreakersTripped : "UDT_EventStatistic";   //  Circuit breakers event statistics
   END_VAR

   VAR
      sUDT_CommonStatus { ExternalAccessible := 'False'; ExternalVisible := 'False'; ExternalWritable := 'False'; S7_SetPoint := 'False'} : "UDT_CommonStatus";   //  Common status structure
      sUDT_CommonStatusOld { ExternalAccessible := 'False'; ExternalVisible := 'False'; ExternalWritable := 'False'; S7_SetPoint := 'False'} : "UDT_CommonStatus";   //  Auxiliary status structure
   END_VAR
   VAR RETAIN
      sUDT_HMIStatus { ExternalAccessible := 'False'; ExternalVisible := 'False'; ExternalWritable := 'False'; S7_SetPoint := 'False'} : "UDT_PowerDistributionPanelStatus";   //  PDP status UDT
   END_VAR
   VAR
      sF_Trig_CircuitBreakerTripped {InstructionName := 'F_TRIG'; LibVersion := '1.0'; ExternalAccessible := 'False'; ExternalVisible := 'False'; ExternalWritable := 'False'; S7_SetPoint := 'False'} : F_TRIG;   //  Fall trigger circuit breaker
      sx_CircuitBreakersStatus { ExternalAccessible := 'False'; ExternalVisible := 'False'; ExternalWritable := 'False'} : Bool;   //  Circuit breakers status
   END_VAR


BEGIN
	(*
	----------------------------------------------------------------------------------------

	Version history:
	Date        | Version   | Author        | Remark
	----------------------------------------------------------------------------------------
	19/09/2019  | 2.0       | C.Leite       | first release TIA 15.1
	15/10/2019  | 2.1       | L.Klar        | Updated status structure
	12/11/2019  | 3.0       | P.Majka       | 3.0 MHS library release TIA 15.1
	25/02/2020  | 3.1       | S. Deulkar    | Modified to update ststus output every cycle
	09/07/2020  | 3.2       | S.Theocharis  | Bug fix in status update. Initialize static status instead output status
	25-02-2021  | 3.3       | M.Kocot       | Added extra circuit breaker to cover all PDP's in one block
	31-03-2021  | 3.4       | H.Rutkowski   | Corrected crosschecked and corrected output write
	02-08-2021  | 3.5       | S. Deulkar    | Masked error if we dont have 24V and profinet okay
	21/02/2023  | 4.0       | F.Baten       | 4.0 Release TIA 17.5
	12/03/2024  | 4.1       | S. Nieswiec   | Updated variable names to current standard
	04/10/2024  | 4.2       | F. Solloch    | Adjust for H&M Cheb
	*)

	REGION 1 - Trigger

	    // Circuit breaker global status
	    #sx_CircuitBreakersStatus := #ix_CircuitBreakerOkF100
	    AND #ix_CircuitBreakerOkF201
	    AND #ix_CircuitBreakerOkF202
	    AND #ix_CircuitBreakerOkF203
	    AND #ix_CircuitBreakerOkF204
	    AND #ix_CircuitBreakerOkF205
	    AND #ix_CircuitBreakerOkF206
	    AND #ix_CircuitBreakerOkF207
	    AND #ix_CircuitBreakerOkF208
	    AND #ix_CircuitBreakerOkF209
	    AND #ix_CircuitBreakerOkF210
	    AND #ix_CircuitBreakerOkF211
	    AND #ix_CircuitBreakerOkF212
	    AND #ix_CircuitBreakerOkF213
	    AND #ix_CircuitBreakerOkF214
	    AND #ix_CircuitBreakerOkF215
	    AND #ix_CircuitBreakerOkF216
	    AND #ix_CircuitBreakerOkF217
	    AND #ix_CircuitBreakerOkF218
	    AND #ix_CircuitBreakerOkF219
	    AND #ix_CircuitBreakerOkF220
	    AND #ix_CircuitBreakerOkF221
	    AND #ix_CircuitBreakerOkF222
	    AND #ix_CircuitBreakerOkF223
	    AND #ix_CircuitBreakerOkF224
	    AND #ix_CircuitBreakerOkF225
	    AND #ix_CircuitBreakerOkF226
	    AND #ix_CircuitBreakerOkF227
	    AND #ix_CircuitBreakerOkF228
	    AND #ix_CircuitBreakerOkF229
	    AND #ix_CircuitBreakerOkF230
	    AND #ix_CircuitBreakerOkF231
	    AND #ix_CircuitBreakerOkF232
	    AND #ix_CircuitBreakerOkF233
	    AND #ix_CircuitBreakerOkF234
	    AND #ix_CircuitBreakerOkF235
	    AND #ix_CircuitBreakerOkF236
	    AND #ix_CircuitBreakerOkF237
	    AND #ix_CircuitBreakerOkF238
	    AND #ix_CircuitBreakerOkF239
	    AND #ix_CircuitBreakerOkF240
	    AND #ix_CircuitBreakerOkF241
	    AND #ix_CircuitBreakerOkF242
	    AND #ix_CircuitBreakerOkF243
	    AND #ix_CircuitBreakerOkF244
	    AND #ix_CircuitBreakerOkF245
	    AND #ix_CircuitBreakerOkF246
	    AND #ix_CircuitBreakerOkF247
	    AND #ix_CircuitBreakerOkF248
	    AND #ix_CircuitBreakerOkF249
	    AND #ix_CircuitBreakerOkF250
	    AND #ix_CircuitBreakerOkF501
	    AND #ix_CircuitBreakerOkF502
	    AND #ix_CircuitBreakerOkF503
	    AND #ix_CircuitBreakerOkF504
	    AND #ix_CircuitBreakerOkF505;

	    // Fall trigger circuit breaker tripped
	    #sF_Trig_CircuitBreakerTripped(CLK := #sx_CircuitBreakersStatus);

	END_REGION

	REGION 2 - Reset faults

	    // All faults are reset when the reset input is true
	    IF #iqUDT_EquipmentControl.Command.Reset
	        OR NOT #ix_ET200Ok
	        OR NOT #ix_24VOk
	    THEN
	        #sUDT_HMIStatus.Specific.CircuitBreakerTrippedF100 := FALSE;
	        #sUDT_HMIStatus.Specific.CircuitBreakerTrippedF201 := FALSE;
	        #sUDT_HMIStatus.Specific.CircuitBreakerTrippedF202 := FALSE;
	        #sUDT_HMIStatus.Specific.CircuitBreakerTrippedF203 := FALSE;
	        #sUDT_HMIStatus.Specific.CircuitBreakerTrippedF204 := FALSE;
	        #sUDT_HMIStatus.Specific.CircuitBreakerTrippedF205 := FALSE;
	        #sUDT_HMIStatus.Specific.CircuitBreakerTrippedF206 := FALSE;
	        #sUDT_HMIStatus.Specific.CircuitBreakerTrippedF207 := FALSE;
	        #sUDT_HMIStatus.Specific.CircuitBreakerTrippedF208 := FALSE;
	        #sUDT_HMIStatus.Specific.CircuitBreakerTrippedF209 := FALSE;
	        #sUDT_HMIStatus.Specific.CircuitBreakerTrippedF210 := FALSE;
	        #sUDT_HMIStatus.Specific.CircuitBreakerTrippedF211 := FALSE;
	        #sUDT_HMIStatus.Specific.CircuitBreakerTrippedF212 := FALSE;
	        #sUDT_HMIStatus.Specific.CircuitBreakerTrippedF213 := FALSE;
	        #sUDT_HMIStatus.Specific.CircuitBreakerTrippedF214 := FALSE;
	        #sUDT_HMIStatus.Specific.CircuitBreakerTrippedF215 := FALSE;
	        #sUDT_HMIStatus.Specific.CircuitBreakerTrippedF216 := FALSE;
	        #sUDT_HMIStatus.Specific.CircuitBreakerTrippedF217 := FALSE;
	        #sUDT_HMIStatus.Specific.CircuitBreakerTrippedF218 := FALSE;
	        #sUDT_HMIStatus.Specific.CircuitBreakerTrippedF219 := FALSE;
	        #sUDT_HMIStatus.Specific.CircuitBreakerTrippedF220 := FALSE;
	        #sUDT_HMIStatus.Specific.CircuitBreakerTrippedF221 := FALSE;
	        #sUDT_HMIStatus.Specific.CircuitBreakerTrippedF222 := FALSE;
	        #sUDT_HMIStatus.Specific.CircuitBreakerTrippedF223 := FALSE;
	        #sUDT_HMIStatus.Specific.CircuitBreakerTrippedF224 := FALSE;
	        #sUDT_HMIStatus.Specific.CircuitBreakerTrippedF225 := FALSE;
	        #sUDT_HMIStatus.Specific.CircuitBreakerTrippedF226 := FALSE;
	        #sUDT_HMIStatus.Specific.CircuitBreakerTrippedF227 := FALSE;
	        #sUDT_HMIStatus.Specific.CircuitBreakerTrippedF228 := FALSE;
	        #sUDT_HMIStatus.Specific.CircuitBreakerTrippedF229 := FALSE;
	        #sUDT_HMIStatus.Specific.CircuitBreakerTrippedF230 := FALSE;
	        #sUDT_HMIStatus.Specific.CircuitBreakerTrippedF231 := FALSE;
	        #sUDT_HMIStatus.Specific.CircuitBreakerTrippedF232 := FALSE;
	        #sUDT_HMIStatus.Specific.CircuitBreakerTrippedF233 := FALSE;
	        #sUDT_HMIStatus.Specific.CircuitBreakerTrippedF234 := FALSE;
	        #sUDT_HMIStatus.Specific.CircuitBreakerTrippedF235 := FALSE;
	        #sUDT_HMIStatus.Specific.CircuitBreakerTrippedF236 := FALSE;
	        #sUDT_HMIStatus.Specific.CircuitBreakerTrippedF237 := FALSE;
	        #sUDT_HMIStatus.Specific.CircuitBreakerTrippedF238 := FALSE;
	        #sUDT_HMIStatus.Specific.CircuitBreakerTrippedF239 := FALSE;
	        #sUDT_HMIStatus.Specific.CircuitBreakerTrippedF240 := FALSE;
	        #sUDT_HMIStatus.Specific.CircuitBreakerTrippedF241 := FALSE;
	        #sUDT_HMIStatus.Specific.CircuitBreakerTrippedF242 := FALSE;
	        #sUDT_HMIStatus.Specific.CircuitBreakerTrippedF243 := FALSE;
	        #sUDT_HMIStatus.Specific.CircuitBreakerTrippedF244 := FALSE;
	        #sUDT_HMIStatus.Specific.CircuitBreakerTrippedF245 := FALSE;
	        #sUDT_HMIStatus.Specific.CircuitBreakerTrippedF246 := FALSE;
	        #sUDT_HMIStatus.Specific.CircuitBreakerTrippedF247 := FALSE;
	        #sUDT_HMIStatus.Specific.CircuitBreakerTrippedF248 := FALSE;
	        #sUDT_HMIStatus.Specific.CircuitBreakerTrippedF249 := FALSE;
	        #sUDT_HMIStatus.Specific.CircuitBreakerTrippedF250 := FALSE;
	        #sUDT_HMIStatus.Specific.CircuitBreakerTrippedF501 := FALSE;
	        #sUDT_HMIStatus.Specific.CircuitBreakerTrippedF502 := FALSE;
	        #sUDT_HMIStatus.Specific.CircuitBreakerTrippedF503 := FALSE;
	        #sUDT_HMIStatus.Specific.CircuitBreakerTrippedF504 := FALSE;
	        #sUDT_HMIStatus.Specific.CircuitBreakerTrippedF505 := FALSE;

	    END_IF;

	END_REGION

	REGION 3 - Faults monitoring

	    // If a circuit breaker is tripped, the state of that is set in HMI Status
	    IF #ix_ET200Ok
	        AND #ix_24VOk
	    THEN

	        IF NOT #sx_CircuitBreakersStatus
	        THEN
	            #sUDT_HMIStatus.Specific.CircuitBreakersTripped := TRUE;
	        END_IF;

	        IF NOT #ix_CircuitBreakerOkF100
	        THEN
	            #sUDT_HMIStatus.Specific.CircuitBreakerTrippedF100 := TRUE;
	        END_IF;

	        IF NOT #ix_CircuitBreakerOkF201
	        THEN
	            #sUDT_HMIStatus.Specific.CircuitBreakerTrippedF201 := TRUE;
	        END_IF;

	        IF NOT #ix_CircuitBreakerOkF202
	        THEN
	            #sUDT_HMIStatus.Specific.CircuitBreakerTrippedF202 := TRUE;
	        END_IF;

	        IF NOT #ix_CircuitBreakerOkF203
	        THEN
	            #sUDT_HMIStatus.Specific.CircuitBreakerTrippedF203 := TRUE;
	        END_IF;

	        IF NOT #ix_CircuitBreakerOkF204
	        THEN
	            #sUDT_HMIStatus.Specific.CircuitBreakerTrippedF204 := TRUE;
	        END_IF;

	        IF NOT #ix_CircuitBreakerOkF205
	        THEN
	            #sUDT_HMIStatus.Specific.CircuitBreakerTrippedF205 := TRUE;
	        END_IF;

	        IF NOT #ix_CircuitBreakerOkF206
	        THEN
	            #sUDT_HMIStatus.Specific.CircuitBreakerTrippedF206 := TRUE;
	        END_IF;

	        IF NOT #ix_CircuitBreakerOkF207
	        THEN
	            #sUDT_HMIStatus.Specific.CircuitBreakerTrippedF207 := TRUE;
	        END_IF;

	        IF NOT #ix_CircuitBreakerOkF208
	        THEN
	            #sUDT_HMIStatus.Specific.CircuitBreakerTrippedF208 := TRUE;
	        END_IF;

	        IF NOT #ix_CircuitBreakerOkF209
	        THEN
	            #sUDT_HMIStatus.Specific.CircuitBreakerTrippedF209 := TRUE;
	        END_IF;

	        IF NOT #ix_CircuitBreakerOkF210
	        THEN
	            #sUDT_HMIStatus.Specific.CircuitBreakerTrippedF210 := TRUE;
	        END_IF;

	        IF NOT #ix_CircuitBreakerOkF211
	        THEN
	            #sUDT_HMIStatus.Specific.CircuitBreakerTrippedF211 := TRUE;
	        END_IF;

	        IF NOT #ix_CircuitBreakerOkF212
	        THEN
	            #sUDT_HMIStatus.Specific.CircuitBreakerTrippedF212 := TRUE;
	        END_IF;

	        IF NOT #ix_CircuitBreakerOkF213
	        THEN
	            #sUDT_HMIStatus.Specific.CircuitBreakerTrippedF213 := TRUE;
	        END_IF;

	        IF NOT #ix_CircuitBreakerOkF214
	        THEN
	            #sUDT_HMIStatus.Specific.CircuitBreakerTrippedF214 := TRUE;
	        END_IF;

	        IF NOT #ix_CircuitBreakerOkF215
	        THEN
	            #sUDT_HMIStatus.Specific.CircuitBreakerTrippedF215 := TRUE;
	        END_IF;

	        IF NOT #ix_CircuitBreakerOkF216
	        THEN
	            #sUDT_HMIStatus.Specific.CircuitBreakerTrippedF216 := TRUE;
	        END_IF;

	        IF NOT #ix_CircuitBreakerOkF217
	        THEN
	            #sUDT_HMIStatus.Specific.CircuitBreakerTrippedF217 := TRUE;
	        END_IF;

	        IF NOT #ix_CircuitBreakerOkF218
	        THEN
	            #sUDT_HMIStatus.Specific.CircuitBreakerTrippedF218 := TRUE;
	        END_IF;

	        IF NOT #ix_CircuitBreakerOkF219
	        THEN
	            #sUDT_HMIStatus.Specific.CircuitBreakerTrippedF219 := TRUE;
	        END_IF;

	        IF NOT #ix_CircuitBreakerOkF220
	        THEN
	            #sUDT_HMIStatus.Specific.CircuitBreakerTrippedF220 := TRUE;
	        END_IF;

	        IF NOT #ix_CircuitBreakerOkF221
	        THEN
	            #sUDT_HMIStatus.Specific.CircuitBreakerTrippedF221 := TRUE;
	        END_IF;

	        IF NOT #ix_CircuitBreakerOkF222
	        THEN
	            #sUDT_HMIStatus.Specific.CircuitBreakerTrippedF222 := TRUE;
	        END_IF;

	        IF NOT #ix_CircuitBreakerOkF223
	        THEN
	            #sUDT_HMIStatus.Specific.CircuitBreakerTrippedF223 := TRUE;
	        END_IF;

	        IF NOT #ix_CircuitBreakerOkF224
	        THEN
	            #sUDT_HMIStatus.Specific.CircuitBreakerTrippedF224 := TRUE;
	        END_IF;

	        IF NOT #ix_CircuitBreakerOkF225
	        THEN
	            #sUDT_HMIStatus.Specific.CircuitBreakerTrippedF225 := TRUE;
	        END_IF;

	        IF NOT #ix_CircuitBreakerOkF226
	        THEN
	            #sUDT_HMIStatus.Specific.CircuitBreakerTrippedF226 := TRUE;
	        END_IF;

	        IF NOT #ix_CircuitBreakerOkF227
	        THEN
	            #sUDT_HMIStatus.Specific.CircuitBreakerTrippedF227 := TRUE;
	        END_IF;

	        IF NOT #ix_CircuitBreakerOkF228
	        THEN
	            #sUDT_HMIStatus.Specific.CircuitBreakerTrippedF228 := TRUE;
	        END_IF;

	        IF NOT #ix_CircuitBreakerOkF229
	        THEN
	            #sUDT_HMIStatus.Specific.CircuitBreakerTrippedF229 := TRUE;
	        END_IF;

	        IF NOT #ix_CircuitBreakerOkF230
	        THEN
	            #sUDT_HMIStatus.Specific.CircuitBreakerTrippedF230 := TRUE;
	        END_IF;

	        IF NOT #ix_CircuitBreakerOkF231
	        THEN
	            #sUDT_HMIStatus.Specific.CircuitBreakerTrippedF231 := TRUE;
	        END_IF;

	        IF NOT #ix_CircuitBreakerOkF232
	        THEN
	            #sUDT_HMIStatus.Specific.CircuitBreakerTrippedF232 := TRUE;
	        END_IF;

	        IF NOT #ix_CircuitBreakerOkF232
	        THEN
	            #sUDT_HMIStatus.Specific.CircuitBreakerTrippedF232 := TRUE;
	        END_IF;

	        IF NOT #ix_CircuitBreakerOkF233
	        THEN
	            #sUDT_HMIStatus.Specific.CircuitBreakerTrippedF233 := TRUE;
	        END_IF;

	        IF NOT #ix_CircuitBreakerOkF234
	        THEN
	            #sUDT_HMIStatus.Specific.CircuitBreakerTrippedF234 := TRUE;
	        END_IF;

	        IF NOT #ix_CircuitBreakerOkF235
	        THEN
	            #sUDT_HMIStatus.Specific.CircuitBreakerTrippedF235 := TRUE;
	        END_IF;

	        IF NOT #ix_CircuitBreakerOkF236
	        THEN
	            #sUDT_HMIStatus.Specific.CircuitBreakerTrippedF236 := TRUE;
	        END_IF;

	        IF NOT #ix_CircuitBreakerOkF237
	        THEN
	            #sUDT_HMIStatus.Specific.CircuitBreakerTrippedF237 := TRUE;
	        END_IF;

	        IF NOT #ix_CircuitBreakerOkF238
	        THEN
	            #sUDT_HMIStatus.Specific.CircuitBreakerTrippedF238 := TRUE;
	        END_IF;

	        IF NOT #ix_CircuitBreakerOkF239
	        THEN
	            #sUDT_HMIStatus.Specific.CircuitBreakerTrippedF239 := TRUE;
	        END_IF;

	        IF NOT #ix_CircuitBreakerOkF240
	        THEN
	            #sUDT_HMIStatus.Specific.CircuitBreakerTrippedF240 := TRUE;
	        END_IF;

	        IF NOT #ix_CircuitBreakerOkF241
	        THEN
	            #sUDT_HMIStatus.Specific.CircuitBreakerTrippedF241 := TRUE;
	        END_IF;

	        IF NOT #ix_CircuitBreakerOkF242
	        THEN
	            #sUDT_HMIStatus.Specific.CircuitBreakerTrippedF242 := TRUE;
	        END_IF;

	        IF NOT #ix_CircuitBreakerOkF243
	        THEN
	            #sUDT_HMIStatus.Specific.CircuitBreakerTrippedF243 := TRUE;
	        END_IF;

	        IF NOT #ix_CircuitBreakerOkF244
	        THEN
	            #sUDT_HMIStatus.Specific.CircuitBreakerTrippedF244 := TRUE;
	        END_IF;

	        IF NOT #ix_CircuitBreakerOkF245
	        THEN
	            #sUDT_HMIStatus.Specific.CircuitBreakerTrippedF245 := TRUE;
	        END_IF;

	        IF NOT #ix_CircuitBreakerOkF246
	        THEN
	            #sUDT_HMIStatus.Specific.CircuitBreakerTrippedF246 := TRUE;
	        END_IF;

	        IF NOT #ix_CircuitBreakerOkF247
	        THEN
	            #sUDT_HMIStatus.Specific.CircuitBreakerTrippedF247 := TRUE;
	        END_IF;

	        IF NOT #ix_CircuitBreakerOkF248
	        THEN
	            #sUDT_HMIStatus.Specific.CircuitBreakerTrippedF248 := TRUE;
	        END_IF;

	        IF NOT #ix_CircuitBreakerOkF249
	        THEN
	            #sUDT_HMIStatus.Specific.CircuitBreakerTrippedF249 := TRUE;
	        END_IF;

	        IF NOT #ix_CircuitBreakerOkF250
	        THEN
	            #sUDT_HMIStatus.Specific.CircuitBreakerTrippedF250 := TRUE;
	        END_IF;

	        IF NOT #ix_CircuitBreakerOkF501
	        THEN
	            #sUDT_HMIStatus.Specific.CircuitBreakerTrippedF501 := TRUE;
	        END_IF;

	        IF NOT #ix_CircuitBreakerOkF502
	        THEN
	            #sUDT_HMIStatus.Specific.CircuitBreakerTrippedF502 := TRUE;
	        END_IF;

	        IF NOT #ix_CircuitBreakerOkF503
	        THEN
	            #sUDT_HMIStatus.Specific.CircuitBreakerTrippedF503 := TRUE;
	        END_IF;

	        IF NOT #ix_CircuitBreakerOkF504
	        THEN
	            #sUDT_HMIStatus.Specific.CircuitBreakerTrippedF504 := TRUE;
	        END_IF;

	        IF NOT #ix_CircuitBreakerOkF505
	        THEN
	            #sUDT_HMIStatus.Specific.CircuitBreakerTrippedF505 := TRUE;
	        END_IF;

	    END_IF;

	END_REGION

	REGION 4 - Status

	    // Set common error to report
	    #sUDT_CommonStatus.Error := #sUDT_HMIStatus.Specific.CircuitBreakerTrippedF100
	    OR #sUDT_HMIStatus.Specific.CircuitBreakerTrippedF201
	    OR #sUDT_HMIStatus.Specific.CircuitBreakerTrippedF202
	    OR #sUDT_HMIStatus.Specific.CircuitBreakerTrippedF203
	    OR #sUDT_HMIStatus.Specific.CircuitBreakerTrippedF204
	    OR #sUDT_HMIStatus.Specific.CircuitBreakerTrippedF205
	    OR #sUDT_HMIStatus.Specific.CircuitBreakerTrippedF206
	    OR #sUDT_HMIStatus.Specific.CircuitBreakerTrippedF207
	    OR #sUDT_HMIStatus.Specific.CircuitBreakerTrippedF208
	    OR #sUDT_HMIStatus.Specific.CircuitBreakerTrippedF209
	    OR #sUDT_HMIStatus.Specific.CircuitBreakerTrippedF210
	    OR #sUDT_HMIStatus.Specific.CircuitBreakerTrippedF211
	    OR #sUDT_HMIStatus.Specific.CircuitBreakerTrippedF212
	    OR #sUDT_HMIStatus.Specific.CircuitBreakerTrippedF213
	    OR #sUDT_HMIStatus.Specific.CircuitBreakerTrippedF214
	    OR #sUDT_HMIStatus.Specific.CircuitBreakerTrippedF215
	    OR #sUDT_HMIStatus.Specific.CircuitBreakerTrippedF216
	    OR #sUDT_HMIStatus.Specific.CircuitBreakerTrippedF217
	    OR #sUDT_HMIStatus.Specific.CircuitBreakerTrippedF218
	    OR #sUDT_HMIStatus.Specific.CircuitBreakerTrippedF219
	    OR #sUDT_HMIStatus.Specific.CircuitBreakerTrippedF220
	    OR #sUDT_HMIStatus.Specific.CircuitBreakerTrippedF221
	    OR #sUDT_HMIStatus.Specific.CircuitBreakerTrippedF222
	    OR #sUDT_HMIStatus.Specific.CircuitBreakerTrippedF223
	    OR #sUDT_HMIStatus.Specific.CircuitBreakerTrippedF224
	    OR #sUDT_HMIStatus.Specific.CircuitBreakerTrippedF225
	    OR #sUDT_HMIStatus.Specific.CircuitBreakerTrippedF225
	    OR #sUDT_HMIStatus.Specific.CircuitBreakerTrippedF226
	    OR #sUDT_HMIStatus.Specific.CircuitBreakerTrippedF227
	    OR #sUDT_HMIStatus.Specific.CircuitBreakerTrippedF228
	    OR #sUDT_HMIStatus.Specific.CircuitBreakerTrippedF229
	    OR #sUDT_HMIStatus.Specific.CircuitBreakerTrippedF230
	    OR #sUDT_HMIStatus.Specific.CircuitBreakerTrippedF231
	    OR #sUDT_HMIStatus.Specific.CircuitBreakerTrippedF232
	    OR #sUDT_HMIStatus.Specific.CircuitBreakerTrippedF233
	    OR #sUDT_HMIStatus.Specific.CircuitBreakerTrippedF234
	    OR #sUDT_HMIStatus.Specific.CircuitBreakerTrippedF235
	    OR #sUDT_HMIStatus.Specific.CircuitBreakerTrippedF236
	    OR #sUDT_HMIStatus.Specific.CircuitBreakerTrippedF237
	    OR #sUDT_HMIStatus.Specific.CircuitBreakerTrippedF238
	    OR #sUDT_HMIStatus.Specific.CircuitBreakerTrippedF239
	    OR #sUDT_HMIStatus.Specific.CircuitBreakerTrippedF240
	    OR #sUDT_HMIStatus.Specific.CircuitBreakerTrippedF241
	    OR #sUDT_HMIStatus.Specific.CircuitBreakerTrippedF242
	    OR #sUDT_HMIStatus.Specific.CircuitBreakerTrippedF243
	    OR #sUDT_HMIStatus.Specific.CircuitBreakerTrippedF244
	    OR #sUDT_HMIStatus.Specific.CircuitBreakerTrippedF245
	    OR #sUDT_HMIStatus.Specific.CircuitBreakerTrippedF246
	    OR #sUDT_HMIStatus.Specific.CircuitBreakerTrippedF247
	    OR #sUDT_HMIStatus.Specific.CircuitBreakerTrippedF248
	    OR #sUDT_HMIStatus.Specific.CircuitBreakerTrippedF249
	    OR #sUDT_HMIStatus.Specific.CircuitBreakerTrippedF250
	    OR #sUDT_HMIStatus.Specific.CircuitBreakerTrippedF501
	    OR #sUDT_HMIStatus.Specific.CircuitBreakerTrippedF502
	    OR #sUDT_HMIStatus.Specific.CircuitBreakerTrippedF503
	    OR #sUDT_HMIStatus.Specific.CircuitBreakerTrippedF504
	    OR #sUDT_HMIStatus.Specific.CircuitBreakerTrippedF505
	    ;

	    // HMI status update
	    IF #sUDT_CommonStatusOld <> #sUDT_CommonStatus                    // update on change
	    THEN

	        // HMI status initialization
	        #sUDT_HMIStatus.Status := 0;

	        // HMI status calculation
	        IF #sUDT_CommonStatus.Error                                    // CB error
	        THEN

	            #sUDT_HMIStatus.Status := "DB_HMIStatusConfiguration".CBError;

	        END_IF;

	        #sUDT_CommonStatusOld := #sUDT_CommonStatus;                  // Copy status to memory
	        #qUDT_Status := #sUDT_CommonStatus;                           // Copy status to output

	    END_IF;

	    #qUDT_HMIStatus := #sUDT_HMIStatus;                           // Copy HMI status to output

	END_REGION

	REGION 5 - Statistics

	    // Statistics is running when at least one circuit breaker is tripped
	    IF #sUDT_HMIStatus.Specific.CircuitBreakersTripped
	        OR #iqUDT_EquipmentControl.Command.ResetData
	    THEN

	        "FC_Statistics"(ix_Reset := #iqUDT_EquipmentControl.Command.ResetData,
	                        ix_Activate := #sUDT_HMIStatus.Specific.CircuitBreakersTripped,
	                        ix_RTrigActivate := #sF_Trig_CircuitBreakerTripped.Q,
	                        iqUDT_Statistics := #iq_CircuitBreakersTripped);

	    END_IF;

	END_REGION

	REGION 6 - Report to control block

	    // Function to manage report between control block and conveyor block
	    "FC_EquipmentReport"(iUDT_Status := #sUDT_CommonStatus,
	                         iqUDT_Control := #iqUDT_EquipmentControl);

	END_REGION

	REGION 7 - Circuit Breake State

	    // State mapping from input to output
	    #qUDT_PdpCbState.CircuitBreakerStateF100 := #ix_CircuitBreakerOkF100;
	    #qUDT_PdpCbState.CircuitBreakerStateF201 := #ix_CircuitBreakerOkF201;
	    #qUDT_PdpCbState.CircuitBreakerStateF202 := #ix_CircuitBreakerOkF202;
	    #qUDT_PdpCbState.CircuitBreakerStateF203 := #ix_CircuitBreakerOkF203;
	    #qUDT_PdpCbState.CircuitBreakerStateF204 := #ix_CircuitBreakerOkF204;
	    #qUDT_PdpCbState.CircuitBreakerStateF205 := #ix_CircuitBreakerOkF205;
	    #qUDT_PdpCbState.CircuitBreakerStateF206 := #ix_CircuitBreakerOkF206;
	    #qUDT_PdpCbState.CircuitBreakerStateF207 := #ix_CircuitBreakerOkF207;
	    #qUDT_PdpCbState.CircuitBreakerStateF208 := #ix_CircuitBreakerOkF208;
	    #qUDT_PdpCbState.CircuitBreakerStateF209 := #ix_CircuitBreakerOkF209;
	    #qUDT_PdpCbState.CircuitBreakerStateF210 := #ix_CircuitBreakerOkF210;
	    #qUDT_PdpCbState.CircuitBreakerStateF211 := #ix_CircuitBreakerOkF211;
	    #qUDT_PdpCbState.CircuitBreakerStateF212 := #ix_CircuitBreakerOkF212;
	    #qUDT_PdpCbState.CircuitBreakerStateF213 := #ix_CircuitBreakerOkF213;
	    #qUDT_PdpCbState.CircuitBreakerStateF214 := #ix_CircuitBreakerOkF214;
	    #qUDT_PdpCbState.CircuitBreakerStateF215 := #ix_CircuitBreakerOkF215;
	    #qUDT_PdpCbState.CircuitBreakerStateF216 := #ix_CircuitBreakerOkF216;
	    #qUDT_PdpCbState.CircuitBreakerStateF217 := #ix_CircuitBreakerOkF217;
	    #qUDT_PdpCbState.CircuitBreakerStateF218 := #ix_CircuitBreakerOkF218;
	    #qUDT_PdpCbState.CircuitBreakerStateF219 := #ix_CircuitBreakerOkF219;
	    #qUDT_PdpCbState.CircuitBreakerStateF220 := #ix_CircuitBreakerOkF220;
	    #qUDT_PdpCbState.CircuitBreakerStateF221 := #ix_CircuitBreakerOkF221;
	    #qUDT_PdpCbState.CircuitBreakerStateF222 := #ix_CircuitBreakerOkF222;
	    #qUDT_PdpCbState.CircuitBreakerStateF223 := #ix_CircuitBreakerOkF223;
	    #qUDT_PdpCbState.CircuitBreakerStateF224 := #ix_CircuitBreakerOkF224;
	    #qUDT_PdpCbState.CircuitBreakerStateF225 := #ix_CircuitBreakerOkF225;
	    #qUDT_PdpCbState.CircuitBreakerStateF226 := #ix_CircuitBreakerOkF226;
	    #qUDT_PdpCbState.CircuitBreakerStateF227 := #ix_CircuitBreakerOkF227;
	    #qUDT_PdpCbState.CircuitBreakerStateF228 := #ix_CircuitBreakerOkF228;
	    #qUDT_PdpCbState.CircuitBreakerStateF229 := #ix_CircuitBreakerOkF229;
	    #qUDT_PdpCbState.CircuitBreakerStateF230 := #ix_CircuitBreakerOkF230;
	    #qUDT_PdpCbState.CircuitBreakerStateF231 := #ix_CircuitBreakerOkF231;
	    #qUDT_PdpCbState.CircuitBreakerStateF232 := #ix_CircuitBreakerOkF232;
	    #qUDT_PdpCbState.CircuitBreakerStateF233 := #ix_CircuitBreakerOkF233;
	    #qUDT_PdpCbState.CircuitBreakerStateF234 := #ix_CircuitBreakerOkF234;
	    #qUDT_PdpCbState.CircuitBreakerStateF235 := #ix_CircuitBreakerOkF235;
	    #qUDT_PdpCbState.CircuitBreakerStateF236 := #ix_CircuitBreakerOkF236;
	    #qUDT_PdpCbState.CircuitBreakerStateF237 := #ix_CircuitBreakerOkF237;
	    #qUDT_PdpCbState.CircuitBreakerStateF238 := #ix_CircuitBreakerOkF238;
	    #qUDT_PdpCbState.CircuitBreakerStateF239 := #ix_CircuitBreakerOkF239;
	    #qUDT_PdpCbState.CircuitBreakerStateF240 := #ix_CircuitBreakerOkF240;
	    #qUDT_PdpCbState.CircuitBreakerStateF241 := #ix_CircuitBreakerOkF241;
	    #qUDT_PdpCbState.CircuitBreakerStateF242 := #ix_CircuitBreakerOkF242;
	    #qUDT_PdpCbState.CircuitBreakerStateF243 := #ix_CircuitBreakerOkF243;
	    #qUDT_PdpCbState.CircuitBreakerStateF244 := #ix_CircuitBreakerOkF244;
	    #qUDT_PdpCbState.CircuitBreakerStateF245 := #ix_CircuitBreakerOkF245;
	    #qUDT_PdpCbState.CircuitBreakerStateF246 := #ix_CircuitBreakerOkF246;
	    #qUDT_PdpCbState.CircuitBreakerStateF247 := #ix_CircuitBreakerOkF247;
	    #qUDT_PdpCbState.CircuitBreakerStateF248 := #ix_CircuitBreakerOkF248;
	    #qUDT_PdpCbState.CircuitBreakerStateF249 := #ix_CircuitBreakerOkF249;
	    #qUDT_PdpCbState.CircuitBreakerStateF250 := #ix_CircuitBreakerOkF250;
	    #qUDT_PdpCbState.CircuitBreakerStateF501 := #ix_CircuitBreakerOkF501;
	    #qUDT_PdpCbState.CircuitBreakerStateF502 := #ix_CircuitBreakerOkF502;
	    #qUDT_PdpCbState.CircuitBreakerStateF503 := #ix_CircuitBreakerOkF503;
	    #qUDT_PdpCbState.CircuitBreakerStateF504 := #ix_CircuitBreakerOkF504;
	    #qUDT_PdpCbState.CircuitBreakerStateF505 := #ix_CircuitBreakerOkF505;


	END_REGION

END_FUNCTION_BLOCK

FUNCTION_BLOCK "FB_ProfiDiag"
TITLE = FB_ProfiDiag
{ S7_Optimized_Access := 'TRUE' }
AUTHOR : MHSE
FAMILY : GeneralSystemFunctions
VERSION : 3.0
// ATTRIBUTES
// AUTO_NUMBER = True
// BLOCK_NUMBER = 25
// END_ATTRIBUTES
//Function block to diagnose Profinet network.
   VAR_INPUT
      iui_LADDR { ExternalAccessible := 'False'; ExternalVisible := 'False'; ExternalWritable := 'False'} : HW_IOSYSTEM;   // Hardware identifier of the PROFINET IO
      ix_ExternalScan { ExternalAccessible := 'False'; ExternalVisible := 'False'; ExternalWritable := 'False'} : Bool;   // External scan
   END_VAR

   VAR_OUTPUT
      qx_ProfinetOk { ExternalAccessible := 'False'; ExternalVisible := 'False'; ExternalWritable := 'False'} : Bool;   // Profinet ok
      qx_Error { ExternalAccessible := 'False'; ExternalVisible := 'False'; ExternalWritable := 'False'} : Bool;   // Collective error output
   END_VAR

   VAR_IN_OUT
      iqUDT_EquipmentControl : "UDT_EquipmentControl";   // Equipment control structure
      iqUDT_PNDiagArray : "UDT_ProfinetNetwork";   // Profinet devices status array
      iqUDT_Statistics : "UDT_ProfiDiagStatistics";   // Statistics structure
   END_VAR

   VAR
      s_GetProjectName {InstructionName := 'Get_Name'; LibVersion := '1.3'; ExternalAccessible := 'False'; ExternalVisible := 'False'; ExternalWritable := 'False'; S7_SetPoint := 'False'} : Get_Name;   // Get name function
      sa_Status { ExternalAccessible := 'False'; ExternalVisible := 'False'; ExternalWritable := 'False'} : Struct   // Status structure
         ErrorCode { ExternalAccessible := 'False'; ExternalVisible := 'False'; ExternalWritable := 'False'} : Struct   // Error code structure
            DeviceState { ExternalAccessible := 'False'; ExternalVisible := 'False'; ExternalWritable := 'False'} : Int;   // Siemens "DeviceState" error code
            GEO2LOG { ExternalAccessible := 'False'; ExternalVisible := 'False'; ExternalWritable := 'False'} : Int;   // Siemens "GEO2LOG" error code
            LOG2GEO { ExternalAccessible := 'False'; ExternalVisible := 'False'; ExternalWritable := 'False'} : Int;   // Siemens "LOG2GEO" error code
            GetName { ExternalAccessible := 'False'; ExternalVisible := 'False'; ExternalWritable := 'False'} : Word;   // Siemens "GetName" error code
         END_STRUCT;
      END_STRUCT;
      sx_PNOK { ExternalAccessible := 'False'; ExternalVisible := 'False'; ExternalWritable := 'False'} : Bool := FALSE;   // Profinet OK
      sx_NewEvent { ExternalAccessible := 'False'; ExternalVisible := 'False'; ExternalWritable := 'False'} : Bool;   // New event
   END_VAR

   VAR_TEMP
      tv_ProfinetGeoAdr {InstructionName := 'GEOADDR'; LibVersion := '1.0'} : GEOADDR;   // Profinet network geo structure
      tv_DeviceGeoAdr {InstructionName := 'GEOADDR'; LibVersion := '1.0'} : GEOADDR;   // Profinet device geo structure
      ta_Configured : Array[0..1024] of Bool;   // Configured devices array
      ta_Exist : Array[0..1024] of Bool;   // Existing devices array
      ta_Error : Array[0..1024] of Bool;   // Devices errors array
      ti_DeviceNr : Int;   // Device number
      ti_NrOfDevicesError : Int;   // Number of devices error
      ti_DiagArraySize : Int;   // Diagnostic array size
   END_VAR

   VAR CONSTANT
      cui_ConfiguredDevicesMode : UInt := 1;   // Scan mode of configured devices
      cui_ExistingDevicesMode : UInt := 4;   // Scan mode of existing devices
      cui_DevicesErrorMode : UInt := 2;   // Scan mode of devices error
      cui_HWType : UInt := 2;   // IO device hardware type
      cui_Area : UInt := 1;   // IO device area
   END_VAR


BEGIN
	(*
	----------------------------------------------------------------------------------------

	Version history:
	Date        | Version   | Author        | Remark
	----------------------------------------------------------------------------------------
	24/05/2019  | 0.1       | K.Pokorski    | first release MHS TIA 15.1
	13/06/2019  | 0.2       | A.Nowak       | Replacement of instruction if for direct write into variable - Region 3
	24/06/2019  | 0.3       | L.Klar        | Status running added
	19/07/2019  | 0.5       | L.Klar        | Status handling changed, output qx_ProfinetOk added
	24/07/2019  | 2.0       | L.Klar        | 2.0 MHS library release TIA 15.1
	14/08/2019  | 2.1       | K.Pokorski    | HW_ID and TIA device project name handling added
	26/08/2019  | 2.2       | K.Pokorski    | Comments adjusted
	20/09/2019  | 2.3       | K.Pokorski    | "UDT_Status" deleted
	04/11/2019  | 2.4       | L.Klar        | Scan profinet and first scan changed from memory bit to DB variable
	12/11/2019  | 3.0       | P.Majka       | 3.0 MHS library release TIA 15.1
	21/02/2023  | 4.0       | F.Baten       | 4.0 Release TIA 17.5
	*)

	REGION 1 – Scan request

	    IF ("DB_Memory".ScanProfinet    // Scan request from diagnostic OB
	        OR "DB_Memory".FirstScan    // First PLC cycle
	        OR #ix_ExternalScan)        // External scan available
	    THEN

	        #sx_PNOK := FALSE;

	    END_IF;

	END_REGION

	REGION 2 – Devices states update

	    // Scan devices, extract device status: configured, exists, error when profinet network not ok
	    IF (NOT #sx_PNOK)       // Profinet needs a scan
	    THEN

	        #sa_Status.ErrorCode.DeviceState := DeviceStates(LADDR := #iui_LADDR,
	                                                         MODE := #cui_ConfiguredDevicesMode,
	                                                         STATE := #ta_Configured);

	        #sa_Status.ErrorCode.DeviceState := DeviceStates(LADDR := #iui_LADDR,
	                                                         MODE := #cui_ExistingDevicesMode,
	                                                         STATE := #ta_Exist);

	        #sa_Status.ErrorCode.DeviceState := DeviceStates(LADDR := #iui_LADDR,
	                                                         MODE := #cui_DevicesErrorMode,
	                                                         STATE := #ta_Error);

	    END_IF;

	END_REGION

	REGION 3 – Devices Statuses update

	    // Move device state to diagnostic structure if network required scan and no error occured during scan
	    IF (NOT #sx_PNOK                                                                                                    // Profinet not ok
	        AND #sa_Status.ErrorCode.DeviceState = 0)                                                                       // "DeviceStates" error free
	    THEN

	        // Initialise reset device errors counter
	        #ti_NrOfDevicesError := 0;

	        // Maximum number of Profinet devices
	        #ti_DiagArraySize := "FC_GetNrOfArrayEl"(iv_Array := #iqUDT_PNDiagArray.DeviceStatus);

	        // A loop operating on Profinet devices
	        FOR #ti_DeviceNr := 0 TO (#ti_DiagArraySize - 1)
	        DO

	            // The device is configured in TIA Portal
	            IF (#ta_Configured[#ti_DeviceNr])                                                                           // Devices configured
	            THEN

	                // Set the device configured status bit in diagnostic structure
	                #iqUDT_PNDiagArray.DeviceStatus[#ti_DeviceNr].DeviceState.Configure := TRUE;

	                // Move device profinet number to diagnostic structure
	                #iqUDT_PNDiagArray.DeviceStatus[#ti_DeviceNr].DeviceState.ProfinetNumber := INT_TO_UINT(#ti_DeviceNr);

	                // Get the Profinet network IOSystem address
	                #sa_Status.ErrorCode.LOG2GEO := LOG2GEO(LADDR := #iui_LADDR, GEOADDR := #tv_ProfinetGeoAdr);

	                // Configuring parameters for extracting the device's HW_ID
	                #tv_DeviceGeoAdr.HWTYPE := #cui_HWType;
	                #tv_DeviceGeoAdr.AREA := #cui_Area;
	                #tv_DeviceGeoAdr.STATION := INT_TO_UINT(#ti_DeviceNr);
	                #tv_DeviceGeoAdr.IOSYSTEM := #tv_ProfinetGeoAdr.IOSYSTEM;

	                // Extracting the device's HW_ID
	                #sa_Status.ErrorCode.GEO2LOG := GEO2LOG(GEOADDR := #tv_DeviceGeoAdr,
	                                                        LADDR => #iqUDT_PNDiagArray.DeviceStatus[#ti_DeviceNr].DeviceState.HW_ID);

	                // Move device's project name to diagnostic structure
	                #s_GetProjectName(LADDR := #iui_LADDR,
	                                  STATION_NR := INT_TO_UINT(#ti_DeviceNr),
	                                  STATUS => #sa_Status.ErrorCode.GetName,
	                                  DATA := #iqUDT_PNDiagArray.DeviceStatus[#ti_DeviceNr].DeviceState.PNDeviceName);

	                // Move device exist state to the Profinet diagnostic structure
	                IF (#ta_Exist[#ti_DeviceNr])                                                                                // Device exist
	                THEN

	                    #iqUDT_PNDiagArray.DeviceStatus[#ti_DeviceNr].DeviceState.Exist := TRUE;

	                ELSE

	                    #iqUDT_PNDiagArray.DeviceStatus[#ti_DeviceNr].DeviceState.Exist := FALSE;

	                    // Increment the number of devices error
	                    #ti_NrOfDevicesError += 1;

	                END_IF;
	                // Move device error state to the Profinet diagnostic structure
	                IF (NOT #ta_Error[#ti_DeviceNr])                                                                            // Device is error free
	                THEN

	                    #iqUDT_PNDiagArray.DeviceStatus[#ti_DeviceNr].DeviceState.Error := FALSE;

	                ELSE

	                    // New error detected
	                    #sx_NewEvent := NOT #iqUDT_PNDiagArray.DeviceStatus[#ti_DeviceNr].DeviceState.Error;

	                    // Statistics handling
	                    IF (#ta_Error[#ti_DeviceNr]                                                                             // Device has error
	                        OR #iqUDT_EquipmentControl.Command.ResetData)                                                      // Reset statistics available
	                    THEN

	                        "FC_Statistics"(ix_Reset := #iqUDT_EquipmentControl.Command.ResetData,
	                                        ix_Activate := #ta_Error[#ti_DeviceNr],
	                                        ix_RTrigActivate := #sx_NewEvent,
	                                        iqUDT_Statistics := #iqUDT_Statistics.DeviceError[#ti_DeviceNr]);

	                    END_IF;

	                    #iqUDT_PNDiagArray.DeviceStatus[#ti_DeviceNr].DeviceState.Error := TRUE;

	                    // Increment number of devices error
	                    #ti_NrOfDevicesError += 1;

	                END_IF;

	                // Reset all diagnostic information if the device is not configured in TIA Portal
	            ELSE

	                #iqUDT_PNDiagArray.DeviceStatus[#ti_DeviceNr].DeviceState.Configure := FALSE;
	                #iqUDT_PNDiagArray.DeviceStatus[#ti_DeviceNr].DeviceState.Exist := FALSE;
	                #iqUDT_PNDiagArray.DeviceStatus[#ti_DeviceNr].DeviceState.Error := FALSE;
	                #iqUDT_PNDiagArray.DeviceStatus[#ti_DeviceNr].DeviceState.HW_ID := 0;
	                #iqUDT_PNDiagArray.DeviceStatus[#ti_DeviceNr].DeviceState.ProfinetNumber := 0;
	                #iqUDT_PNDiagArray.DeviceStatus[#ti_DeviceNr].DeviceState.PNDeviceName := '';

	            END_IF;

	        END_FOR;

	    END_IF;

	END_REGION

	REGION 4 – Profinet OK

	    // Reset profinet error
	    IF (#ti_NrOfDevicesError = 0                        // Number of devices error equal to zero
	        AND (#iqUDT_EquipmentControl.Command.Reset     // Error reset required
	        OR #ix_ExternalScan))                           // External scan active
	    THEN

	        #sx_PNOK := TRUE;

	    END_IF;

	END_REGION

	REGION 5 – Status

	    // Update Profinet ok output status
	    #qx_ProfinetOk := #sx_PNOK;

	    // Create the collective block error bit
	    #qx_Error := #sa_Status.ErrorCode.DeviceState <> 0       // Profinet network error
	    OR #sa_Status.ErrorCode.GEO2LOG <> 0                     // "Geo2Log" standard Siemens block error
	    OR #sa_Status.ErrorCode.LOG2GEO <> 0                     // "Log2Geo" standard Siemens block error
	    OR #sa_Status.ErrorCode.GetName > 16#8000;               // "GetName" standard Siemens block error

	END_REGION
END_FUNCTION_BLOCK

FUNCTION_BLOCK "FB_SlipCompensation"
{ S7_Optimized_Access := 'TRUE' }
VERSION : 0.1
// ATTRIBUTES
// AUTO_NUMBER = True
// BLOCK_NUMBER = 27
// END_ATTRIBUTES
   VAR_INPUT
      IUDT_DowstreamConveyorLength { ExternalAccessible := 'False'; ExternalVisible := 'False'; ExternalWritable := 'False'} : "UDT_ConveyorCommonConfiguration";   //  Configured length of the downstream conveyor
      ii_ConfigurationSlipfactor { ExternalAccessible := 'False'; ExternalVisible := 'False'; ExternalWritable := 'False'} : Int := 0;   //  1-100% slip of the parcel
   END_VAR

   VAR_IN_OUT
      iqUDT_ConveyorInterfaceUpstream : "UDT_ConveyorInterface";   //  Interface structure
      iqUDT_ConveyorInterfaceDownstream : "UDT_ConveyorInterface";   //  Interface structure
      iqUDT_HandShakeUpstream : "UDT_ConveyorHandshake";   //  Upstream handshake structure in forward direction
      iqUDT_HandShakeDownstreamSlip : "UDT_ConveyorHandshake";   //  Downstream handshake structure in forward direction
      iqs_TrackingDataDownstream : Array[*] of Int;   //  Tracking data
   END_VAR

   VAR
      sR_TRIG_TIP {InstructionName := 'R_TRIG'; LibVersion := '1.0'; ExternalAccessible := 'False'; ExternalVisible := 'False'; ExternalWritable := 'False'; S7_SetPoint := 'False'} : R_TRIG;   //  Rising edge trigger TIP signal
      si_MemoryGIN { ExternalAccessible := 'False'; ExternalVisible := 'False'; ExternalWritable := 'False'} : Int;   //  Latest GIN
      si_MemoryParcel { ExternalAccessible := 'False'; ExternalVisible := 'False'; ExternalWritable := 'False'} : Int;   //  Latest Parcellength
      si_CalculatedSlipLength { ExternalAccessible := 'False'; ExternalVisible := 'False'; ExternalWritable := 'False'} : Int;   //  Calculated slip based on lenth of the parcel
      si_ProcessedParcelLength { ExternalAccessible := 'False'; ExternalVisible := 'False'; ExternalWritable := 'False'} : Int;   //  The length of the parcel to be processed
      si_DelayedSlipLength { ExternalAccessible := 'False'; ExternalVisible := 'False'; ExternalWritable := 'False'} : Int;   //  Actual slip counter
      si_LoopCounterWrite { ExternalAccessible := 'False'; ExternalVisible := 'False'; ExternalWritable := 'False'} : Int;   //  LoopCounter write data in tracking array
      sx_ConfigurationError { ExternalAccessible := 'False'; ExternalVisible := 'False'; ExternalWritable := 'False'} : Bool;   //  Error in configuration values
      sx_PositiveSlip { ExternalAccessible := 'False'; ExternalVisible := 'False'; ExternalWritable := 'False'} : Bool;   //  Speed difference is generating positive slip
      sx_NegativeSlip { ExternalAccessible := 'False'; ExternalVisible := 'False'; ExternalWritable := 'False'} : Bool;   //  Speed difference is generating negative slip
   END_VAR


BEGIN
	(*
	----------------------------------------------------------------------------------------

	Version history:
	Date        | Version   | Author        | Remark
	----------------------------------------------------------------------------------------
	30/01/2020  | 3.0       | F.Baten       | first release MHS TIA 15.1
	21/02/2023  | 4.0       | F.Baten       | 4.0 Release TIA 17.5
	*)

	REGION 1 - Configuration error
	    // When slipfactor is less than 1% or bigger than 100% the configuration error is set and passed to both conveyors
	    #sx_ConfigurationError := #ii_ConfigurationSlipfactor > 100 OR #ii_ConfigurationSlipfactor < 1;
	    #iqUDT_ConveyorInterfaceDownstream.ConfigurationError := #sx_ConfigurationError;
	    #iqUDT_ConveyorInterfaceUpstream.ConfigurationError := #sx_ConfigurationError;

	END_REGION

	REGION 2 - Get new gin data
	    IF #iqUDT_HandShakeUpstream.GIN <> 0                                                           // Gin on upstream conveyor
	        AND #iqUDT_HandShakeUpstream.GIN <> #si_MemoryGIN                                          // not equal to previous one
	    THEN
	        #si_MemoryGIN := #iqUDT_HandShakeUpstream.GIN;                                             // Memorise
	        #si_MemoryParcel := "DB_GIN".GIN[#si_MemoryGIN].General.Length;                             // Get the length of this parcel
	        #si_CalculatedSlipLength := REAL_TO_INT((INT_TO_REAL(#si_MemoryParcel) / 100.0) * INT_TO_REAL(#ii_ConfigurationSlipfactor)); // Calculate the distance to generate slip
	        #si_DelayedSlipLength := 0;                                                                 // reset the slipcouter
	        #si_ProcessedParcelLength := #si_MemoryParcel;                                              // copy the memory to the process value
	    END_IF;
	END_REGION

	REGION 3 - Check slip direction
	    // If the speed setpoint of the upstream conveyor is higher than the downstream, the parcel is pushed onto the downstream conveyor
	    // here called "positive slip" the otherway around is then "negative slip".

	    IF #iqUDT_ConveyorInterfaceUpstream.SpeedSetpoint > #iqUDT_ConveyorInterfaceDownstream.SpeedSetpoint
	    THEN
	        #sx_PositiveSlip := TRUE;
	        #sx_NegativeSlip := FALSE;
	    ELSE
	        #sx_PositiveSlip := FALSE;
	        #sx_NegativeSlip := TRUE;
	    END_IF;
	END_REGION

	REGION 4 - Clear upstream NRofPosToShift on own displacement
	    // mimic the working of the tracking for it is not copied to downstream, so with displacement the prositions to shift is decreased
	    IF #iqUDT_HandShakeUpstream.NrOfPosToShift > 0 AND
	        #iqUDT_ConveyorInterfaceUpstream.Displacement > 0
	    THEN
	        #iqUDT_HandShakeUpstream.NrOfPosToShift -= #iqUDT_ConveyorInterfaceUpstream.Displacement;
	        IF #iqUDT_HandShakeUpstream.NrOfPosToShift < 0
	        THEN
	            #iqUDT_HandShakeUpstream.NrOfPosToShift := 0;
	        END_IF;
	    END_IF;
	END_REGION

	REGION 5 - Negative slip handling
	    //  Delay the writing of the data with the slipdistance and then with the displacement
	    //  of the downstream conveyor so the data will catch up because it faster.
	    IF #sx_NegativeSlip
	    THEN

	        REGION 5.1 - Slip delay
	            IF #iqUDT_HandShakeUpstream.TIP                                                        // Transfer is started
	                AND #si_DelayedSlipLength < #si_CalculatedSlipLength                                // Actual slip is not yet reached
	            THEN
	                #si_DelayedSlipLength += #iqUDT_ConveyorInterfaceDownstream.Displacement;          // Increase the slip distance
	            END_IF;
	        END_REGION

	        REGION 5.2 - Pass GIN to downstream
	            IF #si_DelayedSlipLength >= #si_CalculatedSlipLength                                    // The slipdistance is equal or larger to the calculated value
	                AND #si_ProcessedParcelLength > 0                                                   // the lenth of the parcel is not completely processed yet
	            THEN
	                #si_ProcessedParcelLength -= #iqUDT_HandShakeDownstreamSlip.DownstreamDisplacement;    // Decrease the parcel lenth by conveyor displacement

	                #iqUDT_HandShakeDownstreamSlip.NrOfPosToShift := #iqUDT_ConveyorInterfaceDownstream.Displacement; // copy the numbers of positions to shift back to the downstream conveyor
	                #iqUDT_HandShakeDownstreamSlip.GIN := #si_MemoryGIN;
	                IF #si_ProcessedParcelLength < 0                                                    // parcel length too small
	                THEN
	                    #si_ProcessedParcelLength := 0;                                                 // reset length
	                END_IF;
	            END_IF;

	            IF #si_DelayedSlipLength < #si_CalculatedSlipLength                                     // The slipdistance is smaller than the calculated value
	                OR #si_ProcessedParcelLength = 0                                                    // the length of the parcel is processed
	            THEN
	                #iqUDT_HandShakeDownstreamSlip.NrOfPosToShift := 0;                                // reset the value
	                #iqUDT_HandShakeDownstreamSlip.GIN := 0;                                           // clear the GIN
	            END_IF;
	        END_REGION
	    END_IF;
	END_REGION

	REGION 6 - Positive slip handling
	    // Write the data on start of the tip directly in front and then with the displacement of the downstream conveyor
	    // as the parcel is gripped by the conveyor belt.
	    IF #sx_PositiveSlip
	    THEN
	        REGION 6.1 - Parcel entering, write slipped GIN to downstream
	            #sR_TRIG_TIP(CLK := #iqUDT_HandShakeUpstream.TIP
	                         AND (#iqUDT_HandShakeUpstream.GIN <> 0)
	                         AND #iqUDT_HandShakeUpstream.GIN = #si_MemoryGIN);                     // Start of the TIP
	            IF #sR_TRIG_TIP.Q
	            THEN                                                                                // write directly GIN in tracking for the length of the slip
	                FOR #si_LoopCounterWrite := #si_CalculatedSlipLength TO 0 BY -1 DO                      // set the loopcounter
	                    #iqs_TrackingDataDownstream[(#IUDT_DowstreamConveyorLength.Length / 10) - #si_LoopCounterWrite] := #si_MemoryGIN; // Write the GIN from the calculated position to the end
	                END_FOR;
	                #si_ProcessedParcelLength := "DB_GIN".GIN[#si_MemoryGIN].General.Length - #si_CalculatedSlipLength;
	            END_IF;
	        END_REGION

	        REGION 6.2 - Pass remaining GIN to downstream
	            // Calculate the length of the parcel to write GIN
	            // Write the GIN while the parcellength is not '0', reset the values when the parcel is gone but only when in positive slip
	            IF #si_ProcessedParcelLength > 0                                                    // There is still parcellength to process
	            THEN
	                #si_ProcessedParcelLength -= #iqUDT_ConveyorInterfaceDownstream.Displacement;  // decrease the lenth of the value by the downstream displacement
	                IF #si_ProcessedParcelLength < 0                                                // If the length is smaller than '0'
	                THEN
	                    #si_ProcessedParcelLength := 0;                                             // set the value to '0'
	                END_IF;

	                #iqUDT_HandShakeDownstreamSlip.DownstreamDisplacement := #iqUDT_ConveyorInterfaceDownstream.Displacement; // copy the displacement back to the interface
	                #iqUDT_HandShakeDownstreamSlip.GIN := #si_MemoryGIN;                           // copy the gin into the interface
	            END_IF;
	        END_REGION

	        // Parcel was processed, reset values
	        IF #si_ProcessedParcelLength = 0
	        THEN
	            #iqUDT_HandShakeDownstreamSlip.NrOfPosToShift := 0;
	            #iqUDT_HandShakeDownstreamSlip.GIN := 0;
	        END_IF;
	    END_IF;
	END_REGION

